  MoveL 1338 to (-196.6, 429.23, -4.47) mm, rotated rx 180 ry 0 rz -11.91 deg; joints [10.082, -29.328, 80.991, -91.112, 88.613, 140.802]
  MoveL 1339 to (-196.78, 429.13, -4.48) mm, rotated rx -180 ry 0 rz -11.91 deg; joints [10.077, -29.335, 81.007, -91.116, 88.609, 140.811]
  MoveL 1340 to (-196.95, 429.01, -4.47) mm, rotated rx -180 ry 0 rz -11.91 deg; joints [10.072, -29.343, 81.024, -91.12, 88.606, 140.82]
  MoveL 1341 to (-197.13, 428.87, -4.48) mm, rotated rx -180 ry 0 rz -11.91 deg; joints [10.066, -29.352, 81.044, -91.125, 88.604, 140.831]
  MoveL 1342 to (-197.37, 428.65, -4.48) mm, rotated rx 180 ry 0 rz -11.91 deg; joints [10.06, -29.366, 81.073, -91.13, 88.6, 140.847]
  MoveL 1343 to (-197.56, 428.44, -4.48) mm, rotated rx 180 ry 0 rz -11.91 deg; joints [10.055, -29.379, 81.102, -91.134, 88.597, 140.862]
  MoveL 1344 to (-197.72, 428.22, -4.48) mm, rotated rx -180 ry 0 rz -11.91 deg; joints [10.051, -29.391, 81.129, -91.138, 88.595, 140.877]
  MoveL 1345 to (-197.85, 428.01, -4.48) mm, rotated rx -180 ry 0 rz -11.91 deg; joints [10.048, -29.404, 81.157, -91.141, 88.593, 140.892]
  MoveL 1346 to (-197.98, 427.77, -4.48) mm, rotated rx 180 ry 0 rz -11.91 deg; joints [10.045, -29.418, 81.187, -91.143, 88.592, 140.909]
  MoveL 1347 to (-198.08, 427.53, -4.48) mm, rotated rx 180 ry 0 rz -11.91 deg; joints [10.043, -29.432, 81.217, -91.145, 88.591, 140.925]
  MoveL 1348 to (-198.16, 427.29, -4.48) mm, rotated rx 180 ry 0 rz -11.91 deg; joints [10.042, -29.445, 81.246, -91.146, 88.591, 140.94]
  MoveL 1349 to (-198.21, 427.04, -4.47) mm, rotated rx -180 ry 0 rz -11.91 deg; joints [10.042, -29.459, 81.275, -91.147, 88.591, 140.956]
  MoveL 1350 to (-198.25, 426.8, -4.48) mm, rotated rx -180 ry 0 rz -11.91 deg; joints [10.042, -29.472, 81.304, -91.147, 88.591, 140.971]
  MoveL 1351 to (-198.27, 426.56, -4.47) mm, rotated rx -180 ry 0 rz -11.91 deg; joints [10.043, -29.485, 81.332, -91.147, 88.592, 140.986]
  MoveL 1352 to (-198.27, 426.08, -4.48) mm, rotated rx -180 ry 0 rz -11.91 deg; joints [10.045, -29.51, 81.387, -91.146, 88.594, 141.016]
  MoveL 1353 to (-198.27, 425.59, -4.48) mm, rotated rx -180 ry 0 rz -11.91 deg; joints [10.048, -29.536, 81.442, -91.144, 88.597, 141.046]
  MoveL 1354 to (-198.25, 425.35, -4.47) mm, rotated rx -180 ry 0 rz -11.91 deg; joints [10.05, -29.549, 81.47, -91.143, 88.598, 141.061]
  MoveL 1355 to (-198.22, 425.11, -4.47) mm, rotated rx -180 ry 0 rz -11.91 deg; joints [10.053, -29.561, 81.497, -91.141, 88.6, 141.075]
  MoveL 1356 to (-198.16, 424.87, -4.48) mm, rotated rx -180 ry 0 rz -11.91 deg; joints [10.056, -29.573, 81.523, -91.139, 88.602, 141.089]
  MoveL 1357 to (-198.09, 424.63, -4.48) mm, rotated rx 180 ry 0 rz -11.91 deg; joints [10.06, -29.585, 81.549, -91.136, 88.605, 141.103]
  MoveL 1358 to (-197.99, 424.39, -4.48) mm, rotated rx 180 ry 0 rz -11.91 deg; joints [10.065, -29.597, 81.575, -91.133, 88.608, 141.117]
  MoveL 1359 to (-197.87, 424.15, -4.48) mm, rotated rx -180 ry 0 rz -11.91 deg; joints [10.07, -29.609, 81.6, -91.129, 88.612, 141.13]
  MoveL 1360 to (-197.73, 423.93, -4.47) mm, rotated rx -180 ry 0 rz -11.91 deg; joints [10.076, -29.619, 81.622, -91.125, 88.615, 141.142]
  MoveL 1361 to (-197.57, 423.71, -4.48) mm, rotated rx 180 ry 0 rz -11.91 deg; joints [10.083, -29.629, 81.644, -91.12, 88.62, 141.154]
  MoveL 1362 to (-197.38, 423.49, -4.48) mm, rotated rx -180 ry 0 rz -11.91 deg; joints [10.09, -29.639, 81.665, -91.114, 88.625, 141.165]
  MoveL 1363 to (-197.14, 423.27, -4.48) mm, rotated rx -180 ry 0 rz -11.91 deg; joints [10.099, -29.648, 81.685, -91.107, 88.631, 141.176]
  MoveL 1364 to (-196.96, 423.13, -4.48) mm, rotated rx -180 ry 0 rz -11.91 deg; joints [10.106, -29.654, 81.698, -91.102, 88.635, 141.182]
  MoveL 1365 to (-196.78, 423, -4.48) mm, rotated rx 180 ry 0 rz -11.91 deg; joints [10.113, -29.659, 81.708, -91.097, 88.639, 141.188]
  MoveL 1366 to (-196.6, 422.9, -4.48) mm, rotated rx -180 ry 0 rz -11.91 deg; joints [10.119, -29.663, 81.716, -91.092, 88.643, 141.192]
  MoveL 1367 to (-196.42, 422.81, -4.48) mm, rotated rx 180 ry 0 rz -11.91 deg; joints [10.126, -29.666, 81.723, -91.087, 88.647, 141.195]
  MoveL 1368 to (-196.18, 422.71, -4.48) mm, rotated rx -180 ry 0 rz -11.91 deg; joints [10.135, -29.669, 81.729, -91.08, 88.653, 141.199]
  MoveL 1369 to (-195.93, 422.63, -4.47) mm, rotated rx -180 ry 0 rz -11.91 deg; joints [10.143, -29.671, 81.733, -91.073, 88.658, 141.2]
  MoveL 1370 to (-195.69, 422.58, -4.48) mm, rotated rx 180 ry 0 rz -11.91 deg; joints [10.151, -29.671, 81.734, -91.067, 88.663, 141.201]
  MoveL 1371 to (-195.45, 422.54, -4.48) mm, rotated rx -180 ry 0 rz -11.91 deg; joints [10.159, -29.671, 81.733, -91.06, 88.668, 141.2]
  MoveL 1372 to (-195.21, 422.52, -4.48) mm, rotated rx 180 ry 0 rz -11.91 deg; joints [10.167, -29.67, 81.73, -91.054, 88.673, 141.199]
  MoveL 1373 to (-194.97, 422.52, -4.48) mm, rotated rx -180 ry 0 rz -11.91 deg; joints [10.175, -29.668, 81.726, -91.047, 88.678, 141.196]
  Set speed (38.1 mm/s)
  MoveL 1374 to (-194.97, 421.25, -4.48) mm, rotated rx -180 ry 0 rz -11.91 deg; joints [10.183, -29.735, 81.87, -91.043, 88.684, 141.274]
  MoveL 1375 to (-195.61, 421.25, -4.47) mm, rotated rx -180 ry 0 rz -11.91 deg; joints [10.162, -29.74, 81.883, -91.06, 88.671, 141.281]
  Set speed (25.4 mm/s)
  MoveL 1376 to (-195.61, 421.25, -6.84) mm, rotated rx 180 ry 0 rz -11.91 deg; joints [10.163, -29.63, 81.86, -91.062, 88.673, 141.368]
  MoveL 1377 to (-195.61, 421.89, -7.48) mm, rotated rx -180 ry 0 rz -11.91 deg; joints [10.159, -29.567, 81.781, -91.064, 88.67, 141.353]
  Set speed (38.1 mm/s)
  MoveL 1378 to (-194.97, 422.52, -7.47) mm, rotated rx 180 ry 0 rz -11.91 deg; joints [10.176, -29.527, 81.696, -91.05, 88.68, 141.306]
  Set speed (76.2 mm/s)
  MoveL 1379 to (213.41, 422.52, -7.47) mm, rotated rx -180 ry 0 rz -11.91 deg; joints [22.898, -22.659, 66.695, -81.959, 97.664, 133.746]
  MoveL 1380 to (213.89, 422.53, -7.47) mm, rotated rx -180 ry 0 rz -11.91 deg; joints [22.912, -22.646, 66.667, -81.951, 97.676, 133.732]
  MoveL 1381 to (214.13, 422.55, -7.48) mm, rotated rx 180 ry 0 rz -11.91 deg; joints [22.919, -22.638, 66.651, -81.948, 97.682, 133.724]
  MoveL 1382 to (214.37, 422.59, -7.48) mm, rotated rx 180 ry 0 rz -11.91 deg; joints [22.925, -22.629, 66.632, -81.945, 97.688, 133.715]
  MoveL 1383 to (214.61, 422.65, -7.48) mm, rotated rx -180 ry 0 rz -11.91 deg; joints [22.931, -22.619, 66.61, -81.942, 97.694, 133.704]
  MoveL 1384 to (214.85, 422.74, -7.47) mm, rotated rx -180 ry 0 rz -11.91 deg; joints [22.937, -22.608, 66.586, -81.939, 97.7, 133.692]
  MoveL 1385 to (215.09, 422.84, -7.48) mm, rotated rx 180 ry 0 rz -11.91 deg; joints [22.943, -22.595, 66.558, -81.937, 97.706, 133.678]
  MoveL 1386 to (215.34, 422.97, -7.48) mm, rotated rx 180 ry 0 rz -11.91 deg; joints [22.948, -22.58, 66.527, -81.936, 97.712, 133.662]
  MoveL 1387 to (215.58, 423.13, -7.48) mm, rotated rx -180 ry 0 rz -11.91 deg; joints [22.953, -22.564, 66.493, -81.935, 97.718, 133.644]
  MoveL 1388 to (215.82, 423.33, -7.48) mm, rotated rx -180 ry 0 rz -11.91 deg; joints [22.958, -22.546, 66.454, -81.934, 97.724, 133.624]
  MoveL 1389 to (215.96, 423.46, -7.47) mm, rotated rx -180 ry 0 rz -11.91 deg; joints [22.96, -22.533, 66.428, -81.934, 97.728, 133.61]
  MoveL 1390 to (216.09, 423.6, -7.48) mm, rotated rx 180 ry 0 rz -11.91 deg; joints [22.962, -22.522, 66.403, -81.935, 97.731, 133.597]
  MoveL 1391 to (216.2, 423.73, -7.48) mm, rotated rx 180 ry 0 rz -11.91 deg; joints [22.964, -22.51, 66.379, -81.935, 97.734, 133.585]
  MoveL 1392 to (216.3, 423.87, -7.48) mm, rotated rx -180 ry 0 rz -11.91 deg; joints [22.965, -22.499, 66.355, -81.936, 97.737, 133.573]
  MoveL 1393 to (216.39, 424.01, -7.48) mm, rotated rx -180 ry 0 rz -11.91 deg; joints [22.966, -22.488, 66.331, -81.937, 97.739, 133.56]
  MoveL 1394 to (216.47, 424.15, -7.48) mm, rotated rx -180 ry 0 rz -11.91 deg; joints [22.967, -22.477, 66.308, -81.938, 97.741, 133.548]
  MoveL 1395 to (216.6, 424.39, -7.48) mm, rotated rx -180 ry 0 rz -11.91 deg; joints [22.967, -22.459, 66.27, -81.94, 97.745, 133.528]
  MoveL 1396 to (216.69, 424.63, -7.48) mm, rotated rx -180 ry 0 rz -11.91 deg; joints [22.967, -22.441, 66.232, -81.943, 97.747, 133.508]
  MoveL 1397 to (216.77, 424.87, -7.47) mm, rotated rx 180 ry 0 rz -11.91 deg; joints [22.966, -22.424, 66.196, -81.946, 97.749, 133.489]
  MoveL 1398 to (216.82, 425.11, -7.47) mm, rotated rx -180 ry 0 rz -11.91 deg; joints [22.965, -22.407, 66.16, -81.95, 97.751, 133.47]
  MoveL 1399 to (216.86, 425.35, -7.47) mm, rotated rx -180 ry 0 rz -11.91 deg; joints [22.963, -22.391, 66.126, -81.954, 97.752, 133.452]
  MoveL 1400 to (216.88, 425.59, -7.48) mm, rotated rx 180 ry 0 rz -11.91 deg; joints [22.96, -22.376, 66.093, -81.958, 97.753, 133.434]
  MoveL 1401 to (216.88, 426.08, -7.48) mm, rotated rx -180 ry 0 rz -11.91 deg; joints [22.955, -22.345, 66.029, -81.966, 97.753, 133.4]
  MoveL 1402 to (216.88, 427.04, -7.48) mm, rotated rx -180 ry 0 rz -11.91 deg; joints [22.943, -22.284, 65.9, -81.984, 97.754, 133.331]
  MoveL 1403 to (216.86, 427.29, -7.47) mm, rotated rx 180 ry 0 rz -11.91 deg; joints [22.939, -22.269, 65.869, -81.989, 97.754, 133.314]
  MoveL 1404 to (216.83, 427.53, -7.48) mm, rotated rx -180 ry 0 rz -11.91 deg; joints [22.935, -22.255, 65.838, -81.993, 97.754, 133.297]
  MoveL 1405 to (216.78, 427.77, -7.48) mm, rotated rx -180 ry 0 rz -11.91 deg; joints [22.931, -22.241, 65.809, -81.999, 97.753, 133.282]
  MoveL 1406 to (216.71, 428.01, -7.48) mm, rotated rx -180 ry 0 rz -11.91 deg; joints [22.926, -22.228, 65.781, -82.004, 97.751, 133.266]
  MoveL 1407 to (216.63, 428.21, -7.48) mm, rotated rx 180 ry 0 rz -11.91 deg; joints [22.921, -22.217, 65.759, -82.009, 97.749, 133.254]
  MoveL 1408 to (216.54, 428.41, -7.48) mm, rotated rx -180 ry 0 rz -11.91 deg; joints [22.916, -22.207, 65.737, -82.014, 97.747, 133.242]
  MoveL 1409 to (216.43, 428.61, -7.48) mm, rotated rx 180 ry 0 rz -11.91 deg; joints [22.911, -22.197, 65.717, -82.019, 97.745, 133.231]
  MoveL 1410 to (216.3, 428.81, -7.48) mm, rotated rx 180 ry 0 rz -11.91 deg; joints [22.904, -22.188, 65.697, -82.025, 97.742, 133.22]
  MoveL 1411 to (216.16, 428.99, -7.48) mm, rotated rx 180 ry 0 rz -11.91 deg; joints [22.898, -22.18, 65.681, -82.031, 97.738, 133.211]
  MoveL 1412 to (215.99, 429.18, -7.47) mm, rotated rx -180 ry 0 rz -11.91 deg; joints [22.891, -22.173, 65.665, -82.037, 97.735, 133.202]
  MoveL 1413 to (215.78, 429.38, -7.48) mm, rotated rx -180 ry 0 rz -11.91 deg; joints [22.883, -22.165, 65.65, -82.044, 97.729, 133.193]
  MoveL 1414 to (215.57, 429.55, -7.48) mm, rotated rx -180 ry 0 rz -11.91 deg; joints [22.874, -22.16, 65.64, -82.05, 97.724, 133.187]
  MoveL 1415 to (215.39, 429.67, -7.47) mm, rotated rx -180 ry 0 rz -11.91 deg; joints [22.868, -22.157, 65.633, -82.055, 97.72, 133.183]
  MoveL 1416 to (215.21, 429.78, -7.48) mm, rotated rx -180 ry 0 rz -11.91 deg; joints [22.861, -22.155, 65.63, -82.06, 97.716, 133.181]
  MoveL 1417 to (215.02, 429.87, -7.48) mm, rotated rx 180 ry 0 rz -11.91 deg; joints [22.855, -22.154, 65.628, -82.065, 97.711, 133.179]
  MoveL 1418 to (214.84, 429.94, -7.47) mm, rotated rx -180 ry 0 rz -11.91 deg; joints [22.849, -22.154, 65.628, -82.069, 97.707, 133.179]
  MoveL 1419 to (214.61, 430.02, -7.48) mm, rotated rx 180 ry 0 rz -11.91 deg; joints [22.841, -22.156, 65.63, -82.074, 97.701, 133.179]
  MoveL 1420 to (214.37, 430.08, -7.48) mm, rotated rx -180 ry 0 rz -11.91 deg; joints [22.833, -22.158, 65.636, -82.079, 97.695, 133.181]
  MoveL 1421 to (214.13, 430.13, -7.47) mm, rotated rx -180 ry 0 rz -11.91 deg; joints [22.826, -22.162, 65.644, -82.084, 97.689, 133.185]
  MoveL 1422 to (213.89, 430.15, -7.48) mm, rotated rx -180 ry 0 rz -11.91 deg; joints [22.819, -22.166, 65.654, -82.088, 97.683, 133.19]
  MoveL 1423 to (213.41, 430.15, -7.48) mm, rotated rx -180 ry 0 rz -11.91 deg; joints [22.805, -22.179, 65.681, -82.096, 97.671, 133.203]
  MoveL 1424 to (-194.49, 430.15, -7.47) mm, rotated rx 180 ry 0 rz -11.91 deg; joints [10.147, -29.119, 80.811, -91.062, 88.653, 140.83]
  MoveL 1425 to (-195.36, 430.14, -7.48) mm, rotated rx 180 ry 0 rz -11.91 deg; joints [10.118, -29.128, 80.83, -91.084, 88.636, 140.841]
  MoveL 1426 to (-195.58, 430.12, -7.48) mm, rotated rx -180 ry 0 rz -11.91 deg; joints [10.111, -29.131, 80.837, -91.09, 88.631, 140.845]
  MoveL 1427 to (-195.8, 430.08, -7.47) mm, rotated rx 180 ry 0 rz -11.91 deg; joints [10.104, -29.136, 80.847, -91.096, 88.627, 140.85]
  MoveL 1428 to (-196.02, 430.02, -7.48) mm, rotated rx -180 ry 0 rz -11.91 deg; joints [10.097, -29.141, 80.858, -91.101, 88.623, 140.856]
  MoveL 1429 to (-196.24, 429.94, -7.47) mm, rotated rx 180 ry 0 rz -11.91 deg; joints [10.09, -29.147, 80.871, -91.107, 88.619, 140.863]
  MoveL 1430 to (-196.42, 429.87, -7.48) mm, rotated rx -180 ry 0 rz -11.91 deg; joints [10.085, -29.152, 80.884, -91.111, 88.616, 140.87]
  MoveL 1431 to (-196.56, 429.8, -7.48) mm, rotated rx -180 ry 0 rz -11.91 deg; joints [10.08, -29.158, 80.895, -91.115, 88.613, 140.876]
  MoveL 1432 to (-196.71, 429.71, -7.48) mm, rotated rx 180 ry 0 rz -11.91 deg; joints [10.076, -29.163, 80.907, -91.118, 88.61, 140.883]
  MoveL 1433 to (-196.86, 429.62, -7.47) mm, rotated rx 180 ry 0 rz -11.91 deg; joints [10.072, -29.17, 80.921, -91.122, 88.608, 140.891]
  MoveL 1434 to (-197.01, 429.52, -7.47) mm, rotated rx 180 ry 0 rz -11.91 deg; joints [10.067, -29.176, 80.936, -91.125, 88.605, 140.899]
  MoveL 1435 to (-197.15, 429.4, -7.48) mm, rotated rx -180 ry 0 rz -11.91 deg; joints [10.063, -29.184, 80.953, -91.129, 88.603, 140.908]
  MoveL 1436 to (-197.3, 429.27, -7.48) mm, rotated rx -180 ry 0 rz -11.91 deg; joints [10.059, -29.192, 80.971, -91.132, 88.601, 140.918]
  MoveL 1437 to (-197.46, 429.1, -7.48) mm, rotated rx 180 ry 0 rz -11.91 deg; joints [10.055, -29.203, 80.993, -91.136, 88.598, 140.93]
  MoveL 1438 to (-197.6, 428.94, -7.48) mm, rotated rx -180 ry 0 rz -11.91 deg; joints [10.051, -29.213, 81.015, -91.139, 88.596, 140.942]
  MoveL 1439 to (-197.76, 428.71, -7.48) mm, rotated rx -180 ry 0 rz -11.91 deg; joints [10.047, -29.226, 81.045, -91.143, 88.594, 140.958]
  MoveL 1440 to (-197.9, 428.47, -7.48) mm, rotated rx -180 ry 0 rz -11.91 deg; joints [10.044, -29.24, 81.074, -91.146, 88.593, 140.974]
  MoveL 1441 to (-198.01, 428.24, -7.48) mm, rotated rx 180 ry 0 rz -11.91 deg; joints [10.042, -29.253, 81.103, -91.148, 88.591, 140.989]
  MoveL 1442 to (-198.1, 428.01, -7.48) mm, rotated rx 180 ry 0 rz -11.91 deg; joints [10.04, -29.266, 81.132, -91.149, 88.591, 141.005]
  MoveL 1443 to (-198.17, 427.77, -7.48) mm, rotated rx -180 ry 0 rz -11.91 deg; joints [10.039, -29.28, 81.161, -91.151, 88.591, 141.021]
  MoveL 1444 to (-198.23, 427.53, -7.47) mm, rotated rx -180 ry 0 rz -11.91 deg; joints [10.039, -29.293, 81.19, -91.151, 88.591, 141.036]
  MoveL 1445 to (-198.26, 427.29, -7.47) mm, rotated rx -180 ry 0 rz -11.91 deg; joints [10.039, -29.306, 81.218, -91.151, 88.591, 141.051]
  MoveL 1446 to (-198.27, 427.04, -7.47) mm, rotated rx -180 ry 0 rz -11.91 deg; joints [10.04, -29.319, 81.246, -91.151, 88.592, 141.067]
  MoveL 1447 to (-198.27, 426.08, -7.48) mm, rotated rx -180 ry 0 rz -11.91 deg; joints [10.046, -29.37, 81.357, -91.148, 88.597, 141.126]
  MoveL 1448 to (-198.27, 425.59, -7.48) mm, rotated rx 180 ry 0 rz -11.91 deg; joints [10.049, -29.396, 81.412, -91.146, 88.599, 141.156]
  MoveL 1449 to (-198.25, 425.35, -7.48) mm, rotated rx 180 ry 0 rz -11.91 deg; joints [10.051, -29.408, 81.44, -91.145, 88.601, 141.171]
  MoveL 1450 to (-198.22, 425.11, -7.48) mm, rotated rx -180 ry 0 rz -11.91 deg; joints [10.053, -29.421, 81.466, -91.143, 88.603, 141.185]
  MoveL 1451 to (-198.16, 424.87, -7.48) mm, rotated rx -180 ry 0 rz -11.91 deg; joints [10.057, -29.433, 81.493, -91.141, 88.605, 141.199]
  MoveL 1452 to (-198.09, 424.63, -7.48) mm, rotated rx 180 ry 0 rz -11.91 deg; joints [10.061, -29.445, 81.519, -91.138, 88.608, 141.213]
  MoveL 1453 to (-197.99, 424.39, -7.47) mm, rotated rx -180 ry 0 rz -11.91 deg; joints [10.065, -29.457, 81.545, -91.135, 88.611, 141.227]
  MoveL 1454 to (-197.87, 424.15, -7.48) mm, rotated rx 180 ry 0 rz -11.91 deg; joints [10.071, -29.469, 81.57, -91.131, 88.614, 141.24]
  MoveL 1455 to (-197.73, 423.93, -7.48) mm, rotated rx -180 ry 0 rz -11.91 deg; joints [10.077, -29.479, 81.592, -91.127, 88.618, 141.252]
  MoveL 1456 to (-197.57, 423.71, -7.48) mm, rotated rx -180 ry 0 rz -11.91 deg; joints [10.083, -29.489, 81.614, -91.122, 88.622, 141.264]
  MoveL 1457 to (-197.38, 423.49, -7.47) mm, rotated rx -180 ry 0 rz -11.91 deg; joints [10.091, -29.499, 81.635, -91.116, 88.627, 141.275]
  MoveL 1458 to (-197.14, 423.27, -7.47) mm, rotated rx -180 ry 0 rz -11.91 deg; joints [10.1, -29.508, 81.655, -91.109, 88.633, 141.286]
  MoveL 1459 to (-196.96, 423.13, -7.48) mm, rotated rx -180 ry 0 rz -11.91 deg; joints [10.107, -29.514, 81.668, -91.104, 88.637, 141.293]
  MoveL 1460 to (-196.78, 423, -7.47) mm, rotated rx -180 ry 0 rz -11.91 deg; joints [10.113, -29.519, 81.678, -91.099, 88.642, 141.298]
  MoveL 1461 to (-196.6, 422.9, -7.48) mm, rotated rx -180 ry 0 rz -11.91 deg; joints [10.12, -29.523, 81.686, -91.094, 88.646, 141.302]
  MoveL 1462 to (-196.42, 422.81, -7.48) mm, rotated rx 180 ry 0 rz -11.91 deg; joints [10.127, -29.526, 81.693, -91.089, 88.65, 141.306]
  MoveL 1463 to (-196.18, 422.71, -7.48) mm, rotated rx -180 ry 0 rz -11.91 deg; joints [10.135, -29.529, 81.699, -91.082, 88.655, 141.309]
  MoveL 1464 to (-195.93, 422.63, -7.47) mm, rotated rx -180 ry 0 rz -11.91 deg; joints [10.144, -29.53, 81.703, -91.075, 88.66, 141.311]
  MoveL 1465 to (-195.69, 422.58, -7.48) mm, rotated rx -180 ry 0 rz -11.91 deg; joints [10.152, -29.531, 81.704, -91.069, 88.665, 141.311]
  MoveL 1466 to (-195.45, 422.54, -7.48) mm, rotated rx -180 ry 0 rz -11.91 deg; joints [10.16, -29.531, 81.703, -91.062, 88.67, 141.311]
  MoveL 1467 to (-195.21, 422.52, -7.48) mm, rotated rx -180 ry 0 rz -11.91 deg; joints [10.168, -29.53, 81.7, -91.056, 88.675, 141.309]
  MoveL 1468 to (-194.97, 422.52, -7.47) mm, rotated rx 180 ry 0 rz -11.91 deg; joints [10.176, -29.527, 81.696, -91.05, 88.68, 141.306]
  Set speed (38.1 mm/s)
  MoveL 1469 to (-194.97, 421.25, -7.48) mm, rotated rx -180 ry 0 rz -11.91 deg; joints [10.184, -29.594, 81.84, -91.045, 88.686, 141.384]
  MoveL 1470 to (-195.61, 421.25, -7.47) mm, rotated rx -180 ry 0 rz -11.91 deg; joints [10.163, -29.6, 81.853, -91.062, 88.674, 141.392]
  Set speed (25.4 mm/s)
  MoveL 1471 to (-195.61, 421.25, -9.84) mm, rotated rx -180 ry 0 rz -11.91 deg; joints [10.163, -29.489, 81.829, -91.064, 88.675, 141.478]
  MoveL 1472 to (-195.61, 421.89, -10.48) mm, rotated rx -180 ry 0 rz -11.91 deg; joints [10.16, -29.426, 81.75, -91.066, 88.673, 141.463]
  Set speed (38.1 mm/s)
  MoveL 1473 to (-194.97, 422.52, -10.48) mm, rotated rx 180 ry 0 rz -11.91 deg; joints [10.177, -29.387, 81.665, -91.052, 88.683, 141.416]
  Set speed (76.2 mm/s)
  MoveL 1474 to (213.41, 422.52, -10.48) mm, rotated rx -180 ry 0 rz -11.91 deg; joints [22.899, -22.526, 66.66, -81.946, 97.651, 133.844]
  MoveL 1475 to (213.89, 422.53, -10.47) mm, rotated rx -180 ry 0 rz -11.91 deg; joints [22.913, -22.513, 66.632, -81.938, 97.663, 133.83]
  MoveL 1476 to (214.13, 422.55, -10.48) mm, rotated rx -180 ry 0 rz -11.91 deg; joints [22.919, -22.505, 66.616, -81.934, 97.669, 133.822]
  MoveL 1477 to (214.37, 422.59, -10.47) mm, rotated rx 180 ry 0 rz -11.91 deg; joints [22.926, -22.496, 66.597, -81.931, 97.675, 133.813]
  MoveL 1478 to (214.61, 422.65, -10.48) mm, rotated rx -180 ry 0 rz -11.91 deg; joints [22.932, -22.486, 66.575, -81.928, 97.681, 133.802]
  MoveL 1479 to (214.85, 422.74, -10.48) mm, rotated rx -180 ry 0 rz -11.91 deg; joints [22.938, -22.475, 66.551, -81.926, 97.687, 133.79]
  MoveL 1480 to (215.09, 422.84, -10.48) mm, rotated rx -180 ry 0 rz -11.91 deg; joints [22.944, -22.462, 66.523, -81.923, 97.693, 133.776]
  MoveL 1481 to (215.34, 422.97, -10.48) mm, rotated rx -180 ry 0 rz -11.91 deg; joints [22.949, -22.448, 66.493, -81.922, 97.699, 133.76]
  MoveL 1482 to (215.58, 423.13, -10.48) mm, rotated rx 180 ry 0 rz -11.91 deg; joints [22.954, -22.431, 66.458, -81.921, 97.705, 133.742]
  MoveL 1483 to (215.82, 423.33, -10.47) mm, rotated rx -180 ry 0 rz -11.91 deg; joints [22.959, -22.413, 66.419, -81.92, 97.711, 133.722]
  MoveL 1484 to (215.96, 423.46, -10.47) mm, rotated rx -180 ry 0 rz -11.91 deg; joints [22.961, -22.401, 66.393, -81.92, 97.715, 133.708]
  MoveL 1485 to (216.09, 423.6, -10.48) mm, rotated rx -180 ry 0 rz -11.91 deg; joints [22.963, -22.389, 66.368, -81.921, 97.718, 133.695]
  MoveL 1486 to (216.2, 423.73, -10.48) mm, rotated rx 180 ry 0 rz -11.91 deg; joints [22.965, -22.378, 66.344, -81.921, 97.721, 133.683]
  MoveL 1487 to (216.3, 423.87, -10.48) mm, rotated rx -180 ry 0 rz -11.91 deg; joints [22.966, -22.366, 66.32, -81.922, 97.724, 133.67]
  MoveL 1488 to (216.39, 424.01, -10.48) mm, rotated rx -180 ry 0 rz -11.91 deg; joints [22.967, -22.355, 66.296, -81.923, 97.726, 133.658]
  MoveL 1489 to (216.47, 424.15, -10.48) mm, rotated rx -180 ry 0 rz -11.91 deg; joints [22.968, -22.344, 66.273, -81.924, 97.728, 133.646]
  MoveL 1490 to (216.69, 424.27, -10.47) mm, rotated rx -180 ry 0 rz -11.91 deg; joints [22.972, -22.331, 66.245, -81.923, 97.734, 133.631]
  MoveL 1491 to (219.83, 424.27, -10.48) mm, rotated rx -180 ry 0 rz -11.91 deg; joints [23.063, -22.249, 66.068, -81.872, 97.812, 133.546]
  MoveL 1492 to (220.05, 424.15, -10.47) mm, rotated rx -180 ry 0 rz -11.91 deg; joints [23.071, -22.25, 66.071, -81.866, 97.817, 133.548]
  MoveL 1493 to (220.05, 53.41, -10.48) mm, rotated rx 180 ry 0 rz -11.91 deg; joints [28.668, -39.388, 103.529, -74.583, 96.903, 154.267]
  MoveL 1494 to (219.83, 53.18, -10.47) mm, rotated rx -180 ry 0 rz -11.91 deg; joints [28.664, -39.401, 103.558, -74.584, 96.897, 154.283]
  MoveL 1495 to (-199.12, 53.17, -10.48) mm, rotated rx 180 ry 0 rz -11.91 deg; joints [12.81, -44.761, 116.802, -88.93, 89.927, 161.175]
  MoveL 1496 to (-199.7, 53.18, -10.47) mm, rotated rx -180 ry 0 rz -11.91 deg; joints [12.785, -44.765, 116.813, -88.953, 89.92, 161.182]
  MoveL 1497 to (-199.9, 53.41, -10.48) mm, rotated rx 180 ry 0 rz -11.91 deg; joints [12.775, -44.759, 116.797, -88.963, 89.917, 161.172]
  MoveL 1498 to (-199.9, 424.15, -10.48) mm, rotated rx -180 ry 0 rz -11.91 deg; joints [10.004, -29.346, 81.58, -91.187, 88.576, 141.374]
  MoveL 1499 to (-199.7, 424.27, -10.47) mm, rotated rx -180 ry 0 rz -11.91 deg; joints [10.01, -29.338, 81.562, -91.182, 88.58, 141.364]
  MoveL 1500 to (-198.11, 424.27, -10.47) mm, rotated rx -180 ry 0 rz -11.91 deg; joints [10.063, -29.324, 81.53, -91.14, 88.611, 141.346]
  MoveL 1501 to (-197.87, 424.15, -10.48) mm, rotated rx -180 ry 0 rz -11.91 deg; joints [10.071, -29.328, 81.539, -91.133, 88.617, 141.35]
  MoveL 1502 to (-197.73, 423.93, -10.48) mm, rotated rx -180 ry 0 rz -11.91 deg; joints [10.077, -29.338, 81.561, -91.129, 88.621, 141.362]
  MoveL 1503 to (-197.57, 423.71, -10.48) mm, rotated rx -180 ry 0 rz -11.91 deg; joints [10.084, -29.348, 81.583, -91.124, 88.625, 141.374]
  MoveL 1504 to (-197.38, 423.49, -10.48) mm, rotated rx -180 ry 0 rz -11.91 deg; joints [10.092, -29.358, 81.604, -91.118, 88.63, 141.385]
  MoveL 1505 to (-197.14, 423.27, -10.48) mm, rotated rx -180 ry 0 rz -11.91 deg; joints [10.101, -29.368, 81.624, -91.111, 88.636, 141.396]
  MoveL 1506 to (-196.96, 423.13, -10.48) mm, rotated rx -180 ry 0 rz -11.91 deg; joints [10.107, -29.373, 81.637, -91.106, 88.64, 141.402]
  MoveL 1507 to (-196.78, 423, -10.48) mm, rotated rx -180 ry 0 rz -11.91 deg; joints [10.114, -29.378, 81.647, -91.101, 88.644, 141.408]
  MoveL 1508 to (-196.6, 422.9, -10.48) mm, rotated rx 180 ry 0 rz -11.91 deg; joints [10.121, -29.382, 81.655, -91.096, 88.648, 141.412]
  MoveL 1509 to (-196.42, 422.81, -10.48) mm, rotated rx -180 ry 0 rz -11.91 deg; joints [10.127, -29.385, 81.662, -91.091, 88.652, 141.415]
  MoveL 1510 to (-196.18, 422.71, -10.47) mm, rotated rx -180 ry 0 rz -11.91 deg; joints [10.136, -29.388, 81.668, -91.084, 88.658, 141.419]
  MoveL 1511 to (-195.93, 422.63, -10.47) mm, rotated rx -180 ry 0 rz -11.91 deg; joints [10.144, -29.39, 81.672, -91.077, 88.663, 141.421]
  MoveL 1512 to (-195.69, 422.58, -10.48) mm, rotated rx 180 ry 0 rz -11.91 deg; joints [10.153, -29.39, 81.673, -91.071, 88.668, 141.421]
  MoveL 1513 to (-195.45, 422.54, -10.48) mm, rotated rx -180 ry 0 rz -11.91 deg; joints [10.161, -29.39, 81.673, -91.064, 88.673, 141.421]
  MoveL 1514 to (-195.21, 422.52, -10.48) mm, rotated rx 180 ry 0 rz -11.91 deg; joints [10.169, -29.389, 81.67, -91.058, 88.678, 141.419]
  MoveL 1515 to (-194.97, 422.52, -10.48) mm, rotated rx 180 ry 0 rz -11.91 deg; joints [10.177, -29.387, 81.665, -91.052, 88.683, 141.416]
  Set speed (38.1 mm/s)
  MoveL 1516 to (-194.97, 421.25, -10.48) mm, rotated rx -180 ry 0 rz -11.91 deg; joints [10.184, -29.453, 81.81, -91.047, 88.689, 141.494]
  MoveL 1517 to (-195.61, 421.25, -10.48) mm, rotated rx -180 ry 0 rz -11.91 deg; joints [10.163, -29.459, 81.823, -91.064, 88.676, 141.502]
  Set speed (25.4 mm/s)
  MoveL 1518 to (-195.61, 421.25, -12.84) mm, rotated rx -180 ry 0 rz -11.91 deg; joints [10.164, -29.348, 81.798, -91.066, 88.678, 141.588]
  MoveL 1519 to (-195.61, 421.89, -13.48) mm, rotated rx -180 ry 0 rz -11.91 deg; joints [10.16, -29.285, 81.719, -91.068, 88.675, 141.572]
  Set speed (38.1 mm/s)
  MoveL 1520 to (-194.97, 422.52, -13.48) mm, rotated rx 180 ry 0 rz -11.91 deg; joints [10.177, -29.246, 81.633, -91.054, 88.685, 141.526]
  Set speed (76.2 mm/s)
  MoveL 1521 to (213.41, 422.52, -13.48) mm, rotated rx 180 ry 0 rz -11.91 deg; joints [22.9, -22.393, 66.624, -81.932, 97.638, 133.941]
  MoveL 1522 to (213.89, 422.53, -13.47) mm, rotated rx -180 ry 0 rz -11.91 deg; joints [22.914, -22.38, 66.597, -81.924, 97.65, 133.928]
  MoveL 1523 to (214.13, 422.55, -13.47) mm, rotated rx -180 ry 0 rz -11.91 deg; joints [22.92, -22.372, 66.58, -81.92, 97.656, 133.92]
  MoveL 1524 to (214.37, 422.59, -13.47) mm, rotated rx 180 ry 0 rz -11.91 deg; joints [22.927, -22.363, 66.561, -81.917, 97.662, 133.91]
  MoveL 1525 to (214.61, 422.65, -13.48) mm, rotated rx -180 ry 0 rz -11.91 deg; joints [22.933, -22.353, 66.539, -81.914, 97.668, 133.899]
  MoveL 1526 to (214.85, 422.74, -13.47) mm, rotated rx -180 ry 0 rz -11.91 deg; joints [22.939, -22.342, 66.515, -81.912, 97.674, 133.887]
  MoveL 1527 to (215.09, 422.84, -13.48) mm, rotated rx -180 ry 0 rz -11.91 deg; joints [22.945, -22.329, 66.488, -81.91, 97.68, 133.873]
  MoveL 1528 to (215.34, 422.97, -13.48) mm, rotated rx 180 ry 0 rz -11.91 deg; joints [22.95, -22.314, 66.457, -81.908, 97.686, 133.857]
  MoveL 1529 to (215.58, 423.13, -13.47) mm, rotated rx -180 ry 0 rz -11.91 deg; joints [22.955, -22.298, 66.422, -81.907, 97.692, 133.839]
  MoveL 1530 to (215.82, 423.33, -13.47) mm, rotated rx -180 ry 0 rz -11.91 deg; joints [22.96, -22.28, 66.383, -81.907, 97.698, 133.819]
  MoveL 1531 to (215.96, 423.46, -13.48) mm, rotated rx -180 ry 0 rz -11.91 deg; joints [22.962, -22.268, 66.357, -81.907, 97.702, 133.806]
  MoveL 1532 to (216.09, 423.6, -13.48) mm, rotated rx 180 ry 0 rz -11.91 deg; joints [22.964, -22.256, 66.332, -81.907, 97.705, 133.793]
  MoveL 1533 to (216.2, 423.73, -13.47) mm, rotated rx -180 ry 0 rz -11.91 deg; joints [22.966, -22.244, 66.308, -81.908, 97.708, 133.78]
  MoveL 1534 to (216.3, 423.87, -13.48) mm, rotated rx 180 ry 0 rz -11.91 deg; joints [22.967, -22.233, 66.284, -81.908, 97.711, 133.768]
  MoveL 1535 to (216.39, 424.01, -13.48) mm, rotated rx 180 ry 0 rz -11.91 deg; joints [22.968, -22.222, 66.261, -81.909, 97.713, 133.755]
  MoveL 1536 to (216.47, 424.15, -13.47) mm, rotated rx 180 ry 0 rz -11.91 deg; joints [22.968, -22.211, 66.238, -81.911, 97.715, 133.743]
  MoveL 1537 to (216.69, 424.27, -13.47) mm, rotated rx -180 ry 0 rz -11.91 deg; joints [22.973, -22.198, 66.209, -81.909, 97.721, 133.729]
  MoveL 1538 to (219.83, 424.27, -13.48) mm, rotated rx 180 ry 0 rz -11.91 deg; joints [23.064, -22.116, 66.032, -81.858, 97.799, 133.643]
  MoveL 1539 to (220.05, 424.15, -13.47) mm, rotated rx 180 ry 0 rz -11.91 deg; joints [23.072, -22.117, 66.035, -81.852, 97.804, 133.645]
  MoveL 1540 to (220.05, 53.41, -13.48) mm, rotated rx -180 ry 0 rz -11.91 deg; joints [28.669, -39.225, 103.499, -74.566, 96.868, 154.397]
  MoveL 1541 to (219.83, 53.18, -13.47) mm, rotated rx -180 ry 0 rz -11.91 deg; joints [28.665, -39.238, 103.529, -74.567, 96.862, 154.412]
  MoveL 1542 to (-197.29, 53.18, -13.48) mm, rotated rx -180 ry 0 rz -11.91 deg; joints [12.887, -44.563, 116.736, -88.857, 89.949, 161.308]
  MoveL 1543 to (-197.94, 53.18, -13.47) mm, rotated rx -180 ry 0 rz -11.91 deg; joints [12.86, -44.568, 116.748, -88.883, 89.94, 161.315]
  MoveL 1544 to (-198.16, 53.41, -13.47) mm, rotated rx -180 ry 0 rz -11.91 deg; joints [12.848, -44.561, 116.733, -88.894, 89.937, 161.306]
  MoveL 1545 to (-198.16, 424.15, -13.48) mm, rotated rx -180 ry 0 rz -11.91 deg; joints [10.062, -29.19, 81.513, -91.143, 88.614, 141.463]
  MoveL 1546 to (-198.01, 424.27, -13.47) mm, rotated rx -180 ry 0 rz -11.91 deg; joints [10.067, -29.182, 81.496, -91.14, 88.616, 141.454]
  MoveL 1547 to (-197.87, 424.15, -13.47) mm, rotated rx 180 ry 0 rz -11.91 deg; joints [10.072, -29.187, 81.507, -91.135, 88.619, 141.459]
  MoveL 1548 to (-197.73, 423.93, -13.48) mm, rotated rx -180 ry 0 rz -11.91 deg; joints [10.078, -29.197, 81.53, -91.131, 88.623, 141.471]
  MoveL 1549 to (-197.57, 423.71, -13.47) mm, rotated rx -180 ry 0 rz -11.91 deg; joints [10.084, -29.207, 81.551, -91.126, 88.627, 141.483]
  MoveL 1550 to (-197.38, 423.49, -13.47) mm, rotated rx -180 ry 0 rz -11.91 deg; joints [10.092, -29.217, 81.573, -91.12, 88.632, 141.494]
  MoveL 1551 to (-197.22, 423.33, -13.48) mm, rotated rx -180 ry 0 rz -11.91 deg; joints [10.098, -29.224, 81.587, -91.116, 88.636, 141.502]
  MoveL 1552 to (-197.14, 423.27, -13.47) mm, rotated rx -180 ry 0 rz -11.91 deg; joints [10.101, -29.227, 81.593, -91.113, 88.638, 141.505]
  MoveL 1553 to (-196.96, 423.13, -13.48) mm, rotated rx -180 ry 0 rz -11.91 deg; joints [10.108, -29.232, 81.605, -91.108, 88.642, 141.512]
  MoveL 1554 to (-196.78, 423, -13.47) mm, rotated rx -180 ry 0 rz -11.91 deg; joints [10.115, -29.237, 81.615, -91.103, 88.647, 141.517]
  MoveL 1555 to (-196.6, 422.9, -13.48) mm, rotated rx -180 ry 0 rz -11.91 deg; joints [10.121, -29.241, 81.624, -91.098, 88.651, 141.521]
  MoveL 1556 to (-196.42, 422.81, -13.48) mm, rotated rx -180 ry 0 rz -11.91 deg; joints [10.128, -29.244, 81.63, -91.093, 88.655, 141.525]
  MoveL 1557 to (-196.18, 422.71, -13.48) mm, rotated rx 180 ry 0 rz -11.91 deg; joints [10.136, -29.247, 81.637, -91.086, 88.66, 141.528]
  MoveL 1558 to (-195.93, 422.63, -13.48) mm, rotated rx 180 ry 0 rz -11.91 deg; joints [10.145, -29.249, 81.64, -91.079, 88.665, 141.53]
  MoveL 1559 to (-195.69, 422.58, -13.48) mm, rotated rx 180 ry 0 rz -11.91 deg; joints [10.153, -29.249, 81.642, -91.073, 88.67, 141.531]
  MoveL 1560 to (-195.45, 422.54, -13.47) mm, rotated rx -180 ry 0 rz -11.91 deg; joints [10.161, -29.249, 81.641, -91.066, 88.675, 141.53]
  MoveL 1561 to (-195.21, 422.52, -13.48) mm, rotated rx -180 ry 0 rz -11.91 deg; joints [10.169, -29.248, 81.638, -91.06, 88.68, 141.528]
  MoveL 1562 to (-194.97, 422.52, -13.48) mm, rotated rx 180 ry 0 rz -11.91 deg; joints [10.177, -29.246, 81.633, -91.054, 88.685, 141.526]
  Set speed (38.1 mm/s)
  MoveL 1563 to (-194.97, 421.25, -13.48) mm, rotated rx -180 ry 0 rz -11.91 deg; joints [10.185, -29.312, 81.778, -91.049, 88.691, 141.604]
  MoveL 1564 to (-195.61, 421.25, -13.48) mm, rotated rx -180 ry 0 rz -11.91 deg; joints [10.164, -29.318, 81.791, -91.066, 88.678, 141.611]
  Set speed (25.4 mm/s)
  MoveL 1565 to (-195.61, 421.25, -15.84) mm, rotated rx -180 ry 0 rz -11.91 deg; joints [10.165, -29.207, 81.766, -91.068, 88.68, 141.697]
  MoveL 1566 to (-195.61, 421.89, -16.47) mm, rotated rx 180 ry 0 rz -11.91 deg; joints [10.161, -29.144, 81.686, -91.07, 88.678, 141.681]
  Set speed (38.1 mm/s)
  MoveL 1567 to (-194.97, 422.52, -16.48) mm, rotated rx 180 ry 0 rz -11.91 deg; joints [10.178, -29.104, 81.601, -91.056, 88.687, 141.634]
  Set speed (76.2 mm/s)
  MoveL 1568 to (213.41, 422.52, -16.48) mm, rotated rx -180 ry 0 rz -11.91 deg; joints [22.901, -22.259, 66.588, -81.918, 97.625, 134.038]
  MoveL 1569 to (213.89, 422.53, -16.48) mm, rotated rx -180 ry 0 rz -11.91 deg; joints [22.915, -22.246, 66.56, -81.91, 97.637, 134.025]
  MoveL 1570 to (214.13, 422.55, -16.47) mm, rotated rx 180 ry 0 rz -11.91 deg; joints [22.921, -22.238, 66.543, -81.907, 97.643, 134.017]
  MoveL 1571 to (214.37, 422.59, -16.47) mm, rotated rx -180 ry 0 rz -11.91 deg; joints [22.928, -22.23, 66.524, -81.904, 97.649, 134.007]
  MoveL 1572 to (214.61, 422.65, -16.47) mm, rotated rx -180 ry 0 rz -11.91 deg; joints [22.934, -22.219, 66.503, -81.901, 97.655, 133.996]
  MoveL 1573 to (214.85, 422.74, -16.48) mm, rotated rx -180 ry 0 rz -11.91 deg; joints [22.94, -22.208, 66.478, -81.898, 97.661, 133.984]
  MoveL 1574 to (215.09, 422.84, -16.47) mm, rotated rx -180 ry 0 rz -11.91 deg; joints [22.946, -22.195, 66.451, -81.896, 97.667, 133.97]
  MoveL 1575 to (215.34, 422.97, -16.47) mm, rotated rx 180 ry 0 rz -11.91 deg; joints [22.951, -22.181, 66.42, -81.895, 97.673, 133.954]
  MoveL 1576 to (215.58, 423.13, -16.47) mm, rotated rx -180 ry 0 rz -11.91 deg; joints [22.956, -22.165, 66.385, -81.893, 97.679, 133.936]
  MoveL 1577 to (215.82, 423.33, -16.47) mm, rotated rx -180 ry 0 rz -11.91 deg; joints [22.96, -22.146, 66.346, -81.893, 97.685, 133.916]
  MoveL 1578 to (215.96, 423.46, -16.48) mm, rotated rx -180 ry 0 rz -11.91 deg; joints [22.963, -22.134, 66.32, -81.893, 97.689, 133.902]
  MoveL 1579 to (216.09, 423.6, -16.47) mm, rotated rx -180 ry 0 rz -11.91 deg; joints [22.965, -22.122, 66.295, -81.893, 97.692, 133.889]
  MoveL 1580 to (216.2, 423.73, -16.48) mm, rotated rx 180 ry 0 rz -11.91 deg; joints [22.966, -22.111, 66.271, -81.894, 97.695, 133.877]
  MoveL 1581 to (216.3, 423.87, -16.48) mm, rotated rx 180 ry 0 rz -11.91 deg; joints [22.968, -22.1, 66.247, -81.895, 97.698, 133.864]
  MoveL 1582 to (216.39, 424.01, -16.48) mm, rotated rx -180 ry 0 rz -11.91 deg; joints [22.969, -22.089, 66.224, -81.896, 97.7, 133.852]
  MoveL 1583 to (216.47, 424.15, -16.48) mm, rotated rx 180 ry 0 rz -11.91 deg; joints [22.969, -22.078, 66.201, -81.897, 97.702, 133.84]
  MoveL 1584 to (216.69, 424.27, -16.48) mm, rotated rx 180 ry 0 rz -11.91 deg; joints [22.974, -22.065, 66.172, -81.896, 97.708, 133.825]
  MoveL 1585 to (219.83, 424.27, -16.48) mm, rotated rx 180 ry 0 rz -11.91 deg; joints [23.065, -21.982, 65.995, -81.844, 97.786, 133.74]
  MoveL 1586 to (220.05, 424.15, -16.48) mm, rotated rx -180 ry 0 rz -11.91 deg; joints [23.073, -21.984, 65.998, -81.838, 97.791, 133.742]
  MoveL 1587 to (220.05, 53.41, -16.48) mm, rotated rx 180 ry 0 rz -11.91 deg; joints [28.67, -39.062, 103.469, -74.55, 96.833, 154.525]
  MoveL 1588 to (219.83, 53.17, -16.48) mm, rotated rx 180 ry 0 rz -11.91 deg; joints [28.667, -39.075, 103.498, -74.551, 96.827, 154.541]
  MoveL 1589 to (-196.42, 53.17, -16.48) mm, rotated rx -180 ry 0 rz -11.91 deg; joints [12.924, -44.371, 116.688, -88.822, 89.957, 161.451]
  MoveL 1590 to (-196.42, 53.41, -16.47) mm, rotated rx -180 ry 0 rz -11.91 deg; joints [12.921, -44.364, 116.668, -88.824, 89.956, 161.44]
  MoveL 1591 to (-196.42, 422.66, -16.48) mm, rotated rx -180 ry 0 rz -11.91 deg; joints [10.129, -29.111, 81.615, -91.094, 88.658, 141.643]
  MoveL 1592 to (-196.42, 422.81, -16.48) mm, rotated rx 180 ry 0 rz -11.91 deg; joints [10.129, -29.103, 81.598, -91.095, 88.657, 141.634]
  MoveL 1593 to (-196.18, 422.71, -16.48) mm, rotated rx -180 ry 0 rz -11.91 deg; joints [10.137, -29.106, 81.604, -91.088, 88.663, 141.637]
  MoveL 1594 to (-195.93, 422.63, -16.48) mm, rotated rx 180 ry 0 rz -11.91 deg; joints [10.146, -29.107, 81.608, -91.081, 88.668, 141.639]
  MoveL 1595 to (-195.69, 422.58, -16.47) mm, rotated rx -180 ry 0 rz -11.91 deg; joints [10.154, -29.108, 81.609, -91.075, 88.673, 141.64]
  MoveL 1596 to (-195.45, 422.54, -16.48) mm, rotated rx 180 ry 0 rz -11.91 deg; joints [10.162, -29.108, 81.609, -91.068, 88.678, 141.639]
  MoveL 1597 to (-195.21, 422.52, -16.48) mm, rotated rx -180 ry 0 rz -11.91 deg; joints [10.17, -29.107, 81.606, -91.062, 88.683, 141.637]
  MoveL 1598 to (-194.97, 422.52, -16.48) mm, rotated rx 180 ry 0 rz -11.91 deg; joints [10.178, -29.104, 81.601, -91.056, 88.687, 141.634]
  MoveL 1599 to (-164.9, 422.52, -17.52) mm, rotated rx 180 ry 0 rz -11.91 deg; joints [11.168, -28.765, 80.938, -90.266, 89.289, 141.304]
  MoveL 1600 to (213.41, 422.52, -17.52) mm, rotated rx -180 ry 0 rz -11.91 deg; joints [22.901, -22.212, 66.575, -81.914, 97.62, 134.072]
  MoveL 1601 to (213.89, 422.53, -17.52) mm, rotated rx -180 ry 0 rz -11.91 deg; joints [22.915, -22.199, 66.547, -81.906, 97.632, 134.059]
  MoveL 1602 to (214.13, 422.55, -17.53) mm, rotated rx -180 ry 0 rz -11.91 deg; joints [22.922, -22.192, 66.53, -81.902, 97.638, 134.051]
  MoveL 1603 to (214.37, 422.59, -17.53) mm, rotated rx 180 ry 0 rz -11.91 deg; joints [22.928, -22.183, 66.511, -81.899, 97.644, 134.041]
  MoveL 1604 to (214.61, 422.65, -17.52) mm, rotated rx -180 ry 0 rz -11.91 deg; joints [22.934, -22.173, 66.49, -81.896, 97.65, 134.03]
  MoveL 1605 to (214.85, 422.74, -17.53) mm, rotated rx 180 ry 0 rz -11.91 deg; joints [22.94, -22.161, 66.465, -81.894, 97.656, 134.018]
  MoveL 1606 to (215.09, 422.84, -17.53) mm, rotated rx -180 ry 0 rz -11.91 deg; joints [22.946, -22.148, 66.438, -81.891, 97.662, 134.004]
  MoveL 1607 to (215.34, 422.97, -17.52) mm, rotated rx -180 ry 0 rz -11.91 deg; joints [22.951, -22.134, 66.407, -81.89, 97.668, 133.988]
  MoveL 1608 to (215.58, 423.13, -17.53) mm, rotated rx -180 ry 0 rz -11.91 deg; joints [22.956, -22.118, 66.372, -81.889, 97.674, 133.97]
  MoveL 1609 to (215.82, 423.33, -17.53) mm, rotated rx -180 ry 0 rz -11.91 deg; joints [22.961, -22.099, 66.333, -81.888, 97.681, 133.95]
  MoveL 1610 to (215.96, 423.46, -17.52) mm, rotated rx 180 ry 0 rz -11.91 deg; joints [22.963, -22.087, 66.307, -81.888, 97.684, 133.936]
  MoveL 1611 to (216.09, 423.6, -17.53) mm, rotated rx 180 ry 0 rz -11.91 deg; joints [22.965, -22.075, 66.282, -81.889, 97.688, 133.923]
  MoveL 1612 to (216.2, 423.73, -17.53) mm, rotated rx -180 ry 0 rz -11.91 deg; joints [22.967, -22.064, 66.258, -81.889, 97.691, 133.91]
  MoveL 1613 to (216.3, 423.87, -17.52) mm, rotated rx -180 ry 0 rz -11.91 deg; joints [22.968, -22.053, 66.234, -81.89, 97.693, 133.898]
  MoveL 1614 to (216.39, 424.01, -17.53) mm, rotated rx -180 ry 0 rz -11.91 deg; joints [22.969, -22.042, 66.211, -81.891, 97.696, 133.886]
  MoveL 1615 to (216.47, 424.15, -17.53) mm, rotated rx -180 ry 0 rz -11.91 deg; joints [22.97, -22.031, 66.188, -81.892, 97.698, 133.874]
  MoveL 1616 to (216.69, 424.27, -17.52) mm, rotated rx -180 ry 0 rz -11.91 deg; joints [22.975, -22.018, 66.159, -81.891, 97.703, 133.859]
  MoveL 1617 to (219.83, 424.27, -17.52) mm, rotated rx -180 ry 0 rz -11.91 deg; joints [23.065, -21.935, 65.982, -81.84, 97.781, 133.773]
  MoveL 1618 to (220.05, 424.15, -17.53) mm, rotated rx 180 ry 0 rz -11.91 deg; joints [23.073, -21.937, 65.985, -81.834, 97.787, 133.776]
  MoveL 1619 to (220.05, 53.41, -17.52) mm, rotated rx -180 ry 0 rz -11.91 deg; joints [28.671, -39.005, 103.458, -74.544, 96.821, 154.57]
  MoveL 1620 to (219.83, 53.17, -17.53) mm, rotated rx 180 ry 0 rz -11.91 deg; joints [28.667, -39.018, 103.487, -74.545, 96.815, 154.586]
  MoveL 1621 to (-195.15, 53.17, -17.52) mm, rotated rx -180 ry 0 rz -11.91 deg; joints [12.977, -44.297, 116.652, -88.772, 89.972, 161.49]
  MoveL 1622 to (-195.65, 53.17, -17.53) mm, rotated rx -180 ry 0 rz -11.91 deg; joints [12.956, -44.301, 116.662, -88.791, 89.966, 161.496]
  MoveL 1623 to (-195.81, 53.41, -17.52) mm, rotated rx -180 ry 0 rz -11.91 deg; joints [12.947, -44.295, 116.646, -88.8, 89.963, 161.486]
  MoveL 1624 to (-195.81, 422.38, -17.53) mm, rotated rx 180 ry 0 rz -11.91 deg; joints [10.151, -29.07, 81.623, -91.078, 88.672, 141.691]
  MoveL 1625 to (-195.65, 422.57, -17.53) mm, rotated rx -180 ry 0 rz -11.91 deg; joints [10.156, -29.059, 81.598, -91.074, 88.675, 141.678]
  MoveL 1626 to (-195.48, 422.55, -17.53) mm, rotated rx 180 ry 0 rz -11.91 deg; joints [10.161, -29.058, 81.597, -91.07, 88.678, 141.677]
  MoveL 1627 to (-195.32, 422.53, -17.52) mm, rotated rx -180 ry 0 rz -11.91 deg; joints [10.167, -29.058, 81.596, -91.065, 88.681, 141.676]
  MoveL 1628 to (-195.15, 422.52, -17.53) mm, rotated rx -180 ry 0 rz -11.91 deg; joints [10.172, -29.057, 81.593, -91.061, 88.685, 141.675]
  MoveL 1629 to (-194.97, 422.52, -17.53) mm, rotated rx -180 ry 0 rz -11.91 deg; joints [10.178, -29.055, 81.589, -91.056, 88.688, 141.672]
  MoveL 1630 to (-164.9, 422.52, -17.52) mm, rotated rx 180 ry 0 rz -11.91 deg; joints [11.168, -28.765, 80.938, -90.266, 89.289, 141.304]
  Set speed (38.1 mm/s)
  MoveL 1631 to (-164.28, 421.77, -17.53) mm, rotated rx 180 ry 0 rz -11.91 deg; joints [11.194, -28.798, 81.009, -90.246, 89.304, 141.343]
  MoveL 1632 to (-164.81, 418.84, -17.52) mm, rotated rx -180 ry 0 rz -11.91 deg; joints [11.195, -28.957, 81.357, -90.247, 89.306, 141.531]
  MoveL 1633 to (-164.93, 418.21, -16.89) mm, rotated rx -180 ry 0 rz -11.91 deg; joints [11.195, -29.021, 81.438, -90.247, 89.306, 141.548]
  Set speed (100.0 mm/s)
  MoveL 1634 to (-164.93, 418.21, 24.53) mm, rotated rx 180 ry 0 rz -11.91 deg; joints [11.186, -30.941, 81.818, -90.236, 89.294, 140.008]
  MoveL 1635 to (-164.87, 434.05, 24.53) mm, rotated rx 180 ry 0 rz -11.91 deg; joints [11.085, -30.085, 79.996, -90.301, 89.225, 139.043]
  MoveL 1636 to (-164.87, 434.05, -6.52) mm, rotated rx -180 ry 0 rz -11.91 deg; joints [11.092, -28.664, 79.722, -90.311, 89.236, 140.189]
  Set speed (25.4 mm/s)
  MoveL 1637 to (-164.87, 434.05, -9.84) mm, rotated rx 180 ry 0 rz -11.91 deg; joints [11.093, -28.51, 79.688, -90.312, 89.237, 140.309]
  MoveL 1638 to (-164.72, 433.43, -10.48) mm, rotated rx -180 ry 0 rz -11.91 deg; joints [11.102, -28.512, 79.75, -90.306, 89.243, 140.369]
  Set speed (38.1 mm/s)
  MoveL 1639 to (-164.28, 431.48, -10.48) mm, rotated rx 180 ry 0 rz -11.91 deg; joints [11.129, -28.612, 79.966, -90.287, 89.26, 140.485]
  MoveL 1640 to (-164.9, 430.7, -10.48) mm, rotated rx 180 ry 0 rz -11.91 deg; joints [11.113, -28.66, 80.07, -90.299, 89.251, 140.541]
  Set speed (76.2 mm/s)
  MoveL 1641 to (-194.97, 430.7, -10.48) mm, rotated rx -180 ry 0 rz -11.91 deg; joints [10.128, -28.954, 80.726, -91.078, 88.643, 140.91]
  MoveL 1642 to (-202.2, 430.7, -10.48) mm, rotated rx -180 ry 0 rz -11.91 deg; joints [9.89, -29.021, 80.874, -91.267, 88.498, 140.995]
  MoveL 1643 to (-203.17, 430.7, -10.48) mm, rotated rx -180 ry 0 rz -11.91 deg; joints [9.858, -29.029, 80.894, -91.293, 88.478, 141.006]
  MoveL 1644 to (-203.41, 430.69, -10.47) mm, rotated rx -180 ry 0 rz -11.91 deg; joints [9.851, -29.032, 80.901, -91.299, 88.474, 141.01]
  MoveL 1645 to (-203.65, 430.65, -10.48) mm, rotated rx -180 ry 0 rz -11.91 deg; joints [9.843, -29.037, 80.91, -91.305, 88.469, 141.015]
  MoveL 1646 to (-203.89, 430.6, -10.48) mm, rotated rx 180 ry 0 rz -11.91 deg; joints [9.835, -29.042, 80.921, -91.311, 88.464, 141.021]
  MoveL 1647 to (-204.13, 430.52, -10.47) mm, rotated rx -180 ry 0 rz -11.91 deg; joints [9.828, -29.048, 80.934, -91.317, 88.46, 141.029]
  MoveL 1648 to (-204.42, 430.43, -10.48) mm, rotated rx -180 ry 0 rz -11.91 deg; joints [9.819, -29.055, 80.951, -91.325, 88.455, 141.038]
  MoveL 1649 to (-204.57, 430.37, -10.47) mm, rotated rx -180 ry 0 rz -11.91 deg; joints [9.814, -29.06, 80.96, -91.328, 88.452, 141.043]
  MoveL 1650 to (-204.72, 430.31, -10.47) mm, rotated rx 180 ry 0 rz -11.91 deg; joints [9.81, -29.064, 80.971, -91.332, 88.449, 141.049]
  MoveL 1651 to (-204.86, 430.23, -10.48) mm, rotated rx 180 ry 0 rz -11.91 deg; joints [9.805, -29.07, 80.982, -91.336, 88.447, 141.055]
  MoveL 1652 to (-205.01, 430.15, -10.47) mm, rotated rx -180 ry 0 rz -11.91 deg; joints [9.801, -29.075, 80.995, -91.339, 88.444, 141.062]
  MoveL 1653 to (-205.16, 430.05, -10.48) mm, rotated rx -180 ry 0 rz -11.91 deg; joints [9.797, -29.082, 81.009, -91.343, 88.442, 141.07]
  MoveL 1654 to (-205.3, 429.94, -10.48) mm, rotated rx -180 ry 0 rz -11.91 deg; joints [9.792, -29.089, 81.024, -91.346, 88.439, 141.078]
  MoveL 1655 to (-205.53, 429.75, -10.48) mm, rotated rx 180 ry 0 rz -11.91 deg; joints [9.786, -29.101, 81.051, -91.352, 88.436, 141.093]
  MoveL 1656 to (-205.75, 429.52, -10.48) mm, rotated rx 180 ry 0 rz -11.91 deg; joints [9.78, -29.115, 81.082, -91.357, 88.433, 141.11]
  MoveL 1657 to (-205.92, 429.3, -10.48) mm, rotated rx -180 ry 0 rz -11.91 deg; joints [9.776, -29.128, 81.11, -91.361, 88.43, 141.125]
  MoveL 1658 to (-206.06, 429.09, -10.48) mm, rotated rx -180 ry 0 rz -11.91 deg; joints [9.772, -29.141, 81.137, -91.364, 88.428, 141.14]
  MoveL 1659 to (-206.14, 428.96, -10.48) mm, rotated rx -180 ry 0 rz -11.91 deg; joints [9.771, -29.149, 81.155, -91.366, 88.428, 141.149]
  MoveL 1660 to (-206.21, 428.82, -10.48) mm, rotated rx -180 ry 0 rz -11.91 deg; joints [9.769, -29.156, 81.171, -91.367, 88.427, 141.158]
  MoveL 1661 to (-206.27, 428.69, -10.48) mm, rotated rx -180 ry 0 rz -11.91 deg; joints [9.768, -29.164, 81.188, -91.368, 88.426, 141.167]
  MoveL 1662 to (-206.32, 428.55, -10.48) mm, rotated rx -180 ry 0 rz -11.91 deg; joints [9.767, -29.172, 81.205, -91.369, 88.426, 141.176]
  MoveL 1663 to (-206.37, 428.42, -10.47) mm, rotated rx -180 ry 0 rz -11.91 deg; joints [9.766, -29.179, 81.221, -91.37, 88.426, 141.185]
  MoveL 1664 to (-206.41, 428.28, -10.47) mm, rotated rx -180 ry 0 rz -11.91 deg; joints [9.765, -29.187, 81.237, -91.371, 88.426, 141.194]
  MoveL 1665 to (-206.47, 428.01, -10.47) mm, rotated rx -180 ry 0 rz -11.91 deg; joints [9.765, -29.202, 81.27, -91.372, 88.426, 141.211]
  MoveL 1666 to (-206.5, 427.77, -10.48) mm, rotated rx 180 ry 0 rz -11.91 deg; joints [9.765, -29.215, 81.298, -91.372, 88.426, 141.227]
  MoveL 1667 to (-206.52, 427.53, -10.47) mm, rotated rx -180 ry 0 rz -11.91 deg; joints [9.766, -29.228, 81.326, -91.372, 88.427, 141.242]
  MoveL 1668 to (-206.52, 427.04, -10.48) mm, rotated rx 180 ry 0 rz -11.91 deg; joints [9.769, -29.253, 81.381, -91.37, 88.429, 141.272]
  MoveL 1669 to (-206.52, 50.21, -10.47) mm, rotated rx 180 ry 0 rz -11.91 deg; joints [12.529, -44.912, 117.182, -89.198, 89.838, 161.403]
  MoveL 1670 to (-206.51, 49.73, -10.47) mm, rotated rx -180 ry 0 rz -11.91 deg; joints [12.534, -44.927, 117.221, -89.193, 89.839, 161.427]
  MoveL 1671 to (-206.48, 49.48, -10.47) mm, rotated rx -180 ry 0 rz -11.91 deg; joints [12.538, -44.935, 117.241, -89.189, 89.84, 161.438]
  MoveL 1672 to (-206.43, 49.24, -10.47) mm, rotated rx -180 ry 0 rz -11.91 deg; joints [12.542, -44.943, 117.26, -89.185, 89.841, 161.45]
  MoveL 1673 to (-206.37, 49.02, -10.48) mm, rotated rx -180 ry 0 rz -11.91 deg; joints [12.547, -44.95, 117.277, -89.181, 89.842, 161.46]
  MoveL 1674 to (-206.28, 48.8, -10.48) mm, rotated rx -180 ry 0 rz -11.91 deg; joints [12.553, -44.957, 117.293, -89.176, 89.844, 161.47]
  MoveL 1675 to (-206.18, 48.57, -10.48) mm, rotated rx 180 ry 0 rz -11.91 deg; joints [12.559, -44.963, 117.31, -89.17, 89.846, 161.48]
  MoveL 1676 to (-206.06, 48.35, -10.48) mm, rotated rx 180 ry 0 rz -11.91 deg; joints [12.566, -44.97, 117.326, -89.163, 89.848, 161.489]
  MoveL 1677 to (-205.98, 48.22, -10.47) mm, rotated rx -180 ry 0 rz -11.91 deg; joints [12.571, -44.973, 117.335, -89.158, 89.849, 161.495]
  MoveL 1678 to (-205.88, 48.09, -10.48) mm, rotated rx 180 ry 0 rz -11.91 deg; joints [12.576, -44.977, 117.344, -89.153, 89.851, 161.5]
  MoveL 1679 to (-205.78, 47.96, -10.48) mm, rotated rx 180 ry 0 rz -11.91 deg; joints [12.582, -44.981, 117.353, -89.148, 89.852, 161.505]
  MoveL 1680 to (-205.66, 47.83, -10.48) mm, rotated rx -180 ry 0 rz -11.91 deg; joints [12.588, -44.984, 117.361, -89.142, 89.854, 161.51]
  MoveL 1681 to (-205.51, 47.67, -10.48) mm, rotated rx 180 ry 0 rz -11.91 deg; joints [12.596, -44.988, 117.371, -89.135, 89.856, 161.516]
  MoveL 1682 to (-205.35, 47.54, -10.48) mm, rotated rx -180 ry 0 rz -11.91 deg; joints [12.604, -44.992, 117.38, -89.127, 89.859, 161.521]
  MoveL 1683 to (-205.19, 47.42, -10.47) mm, rotated rx -180 ry 0 rz -11.91 deg; joints [12.611, -44.995, 117.387, -89.12, 89.861, 161.525]
  MoveL 1684 to (-205.03, 47.31, -10.48) mm, rotated rx -180 ry 0 rz -11.91 deg; joints [12.619, -44.997, 117.392, -89.113, 89.863, 161.529]
  MoveL 1685 to (-204.81, 47.18, -10.48) mm, rotated rx 180 ry 0 rz -11.91 deg; joints [12.629, -45, 117.399, -89.103, 89.866, 161.532]
  MoveL 1686 to (-204.58, 47.08, -10.47) mm, rotated rx 180 ry 0 rz -11.91 deg; joints [12.64, -45.001, 117.403, -89.093, 89.869, 161.535]
  MoveL 1687 to (-204.36, 46.99, -10.47) mm, rotated rx -180 ry 0 rz -11.91 deg; joints [12.65, -45.003, 117.406, -89.083, 89.872, 161.537]
  MoveL 1688 to (-204.13, 46.92, -10.48) mm, rotated rx -180 ry 0 rz -11.91 deg; joints [12.66, -45.003, 117.407, -89.073, 89.875, 161.538]
  MoveL 1689 to (-203.89, 46.87, -10.47) mm, rotated rx 180 ry 0 rz -11.91 deg; joints [12.671, -45.003, 117.407, -89.063, 89.879, 161.537]
  MoveL 1690 to (-203.65, 46.84, -10.47) mm, rotated rx 180 ry 0 rz -11.91 deg; joints [12.681, -45.003, 117.405, -89.053, 89.882, 161.536]
  MoveL 1691 to (-203.41, 46.83, -10.48) mm, rotated rx -180 ry 0 rz -11.91 deg; joints [12.691, -45.002, 117.402, -89.044, 89.885, 161.534]
  MoveL 1692 to (-203.17, 46.83, -10.47) mm, rotated rx -180 ry 0 rz -11.91 deg; joints [12.701, -45, 117.398, -89.034, 89.888, 161.531]
  MoveL 1693 to (222.09, 46.82, -10.48) mm, rotated rx 180 ry 0 rz -11.91 deg; joints [28.858, -39.583, 103.974, -74.38, 96.915, 154.532]
  MoveL 1694 to (223.29, 46.83, -10.48) mm, rotated rx -180 ry 0 rz -11.91 deg; joints [28.898, -39.561, 103.92, -74.346, 96.941, 154.506]
  MoveL 1695 to (223.53, 46.84, -10.48) mm, rotated rx 180 ry 0 rz -11.91 deg; joints [28.906, -39.555, 103.908, -74.34, 96.946, 154.5]
  MoveL 1696 to (223.77, 46.87, -10.47) mm, rotated rx 180 ry 0 rz -11.91 deg; joints [28.914, -39.55, 103.895, -74.334, 96.951, 154.494]
  MoveL 1697 to (224.01, 46.92, -10.47) mm, rotated rx -180 ry 0 rz -11.91 deg; joints [28.921, -39.543, 103.88, -74.328, 96.956, 154.486]
  MoveL 1698 to (224.24, 46.99, -10.47) mm, rotated rx -180 ry 0 rz -11.91 deg; joints [28.927, -39.537, 103.864, -74.324, 96.961, 154.478]
  MoveL 1699 to (224.46, 47.08, -10.48) mm, rotated rx 180 ry 0 rz -11.91 deg; joints [28.933, -39.529, 103.847, -74.319, 96.967, 154.47]
  MoveL 1700 to (224.69, 47.18, -10.48) mm, rotated rx 180 ry 0 rz -11.91 deg; joints [28.939, -39.521, 103.828, -74.315, 96.972, 154.46]
  MoveL 1701 to (224.92, 47.31, -10.48) mm, rotated rx 180 ry 0 rz -11.91 deg; joints [28.944, -39.513, 103.808, -74.312, 96.977, 154.449]
  MoveL 1702 to (225.07, 47.42, -10.47) mm, rotated rx -180 ry 0 rz -11.91 deg; joints [28.947, -39.506, 103.792, -74.31, 96.981, 154.441]
  MoveL 1703 to (225.23, 47.54, -10.47) mm, rotated rx -180 ry 0 rz -11.91 deg; joints [28.95, -39.499, 103.775, -74.308, 96.985, 154.432]
  MoveL 1704 to (225.39, 47.67, -10.48) mm, rotated rx 180 ry 0 rz -11.91 deg; joints [28.953, -39.491, 103.757, -74.307, 96.989, 154.422]
  MoveL 1705 to (225.55, 47.83, -10.47) mm, rotated rx 180 ry 0 rz -11.91 deg; joints [28.955, -39.482, 103.737, -74.306, 96.993, 154.411]
  MoveL 1706 to (225.66, 47.96, -10.47) mm, rotated rx 180 ry 0 rz -11.91 deg; joints [28.957, -39.475, 103.721, -74.306, 96.996, 154.403]
  MoveL 1707 to (225.77, 48.09, -10.48) mm, rotated rx -180 ry 0 rz -11.91 deg; joints [28.958, -39.469, 103.706, -74.306, 96.999, 154.395]
  MoveL 1708 to (225.86, 48.22, -10.48) mm, rotated rx 180 ry 0 rz -11.91 deg; joints [28.959, -39.462, 103.691, -74.306, 97.001, 154.387]
  MoveL 1709 to (225.94, 48.35, -10.48) mm, rotated rx -180 ry 0 rz -11.91 deg; joints [28.959, -39.456, 103.677, -74.307, 97.004, 154.379]
  MoveL 1710 to (226.07, 48.57, -10.48) mm, rotated rx 180 ry 0 rz -11.91 deg; joints [28.959, -39.446, 103.653, -74.309, 97.007, 154.366]
  MoveL 1711 to (226.17, 48.8, -10.48) mm, rotated rx -180 ry 0 rz -11.91 deg; joints [28.958, -39.436, 103.631, -74.311, 97.01, 154.353]
  MoveL 1712 to (226.25, 49.02, -10.47) mm, rotated rx -180 ry 0 rz -11.91 deg; joints [28.957, -39.427, 103.609, -74.314, 97.013, 154.341]
  MoveL 1713 to (226.31, 49.24, -10.47) mm, rotated rx 180 ry 0 rz -11.91 deg; joints [28.955, -39.418, 103.588, -74.317, 97.015, 154.329]
  MoveL 1714 to (226.36, 49.48, -10.47) mm, rotated rx -180 ry 0 rz -11.91 deg; joints [28.952, -39.408, 103.566, -74.321, 97.018, 154.317]
  MoveL 1715 to (226.39, 49.73, -10.48) mm, rotated rx -180 ry 0 rz -11.91 deg; joints [28.948, -39.399, 103.545, -74.325, 97.019, 154.305]
  MoveL 1716 to (226.4, 50.21, -10.48) mm, rotated rx -180 ry 0 rz -11.91 deg; joints [28.94, -39.382, 103.505, -74.336, 97.022, 154.282]
  MoveL 1717 to (226.4, 427.53, -10.48) mm, rotated rx -180 ry 0 rz -11.91 deg; joints [23.212, -21.867, 65.255, -81.826, 97.98, 133.131]
  MoveL 1718 to (226.39, 427.77, -10.48) mm, rotated rx 180 ry 0 rz -11.91 deg; joints [23.208, -21.852, 65.223, -81.831, 97.98, 133.113]
  MoveL 1719 to (226.37, 428.01, -10.47) mm, rotated rx 180 ry 0 rz -11.91 deg; joints [23.205, -21.837, 65.192, -81.836, 97.979, 133.097]
  MoveL 1720 to (226.34, 428.16, -10.47) mm, rotated rx 180 ry 0 rz -11.91 deg; joints [23.202, -21.829, 65.174, -81.839, 97.979, 133.087]
  MoveL 1721 to (226.31, 428.3, -10.47) mm, rotated rx -180 ry 0 rz -11.91 deg; joints [23.199, -21.82, 65.157, -81.842, 97.978, 133.077]
  MoveL 1722 to (226.27, 428.45, -10.47) mm, rotated rx -180 ry 0 rz -11.91 deg; joints [23.196, -21.812, 65.139, -81.845, 97.977, 133.068]
  MoveL 1723 to (226.22, 428.59, -10.48) mm, rotated rx 180 ry 0 rz -11.91 deg; joints [23.193, -21.804, 65.122, -81.849, 97.976, 133.059]
  MoveL 1724 to (226.16, 428.74, -10.48) mm, rotated rx 180 ry 0 rz -11.91 deg; joints [23.19, -21.796, 65.106, -81.852, 97.975, 133.05]
  MoveL 1725 to (226.1, 428.89, -10.47) mm, rotated rx -180 ry 0 rz -11.91 deg; joints [23.186, -21.789, 65.09, -81.856, 97.974, 133.041]
  MoveL 1726 to (226.03, 429.03, -10.48) mm, rotated rx -180 ry 0 rz -11.91 deg; joints [23.182, -21.781, 65.075, -81.86, 97.972, 133.033]
  MoveL 1727 to (225.94, 429.18, -10.48) mm, rotated rx -180 ry 0 rz -11.91 deg; joints [23.178, -21.774, 65.06, -81.864, 97.97, 133.024]
  MoveL 1728 to (225.82, 429.37, -10.48) mm, rotated rx 180 ry 0 rz -11.91 deg; joints [23.172, -21.765, 65.041, -81.87, 97.967, 133.014]
  MoveL 1729 to (225.67, 429.56, -10.48) mm, rotated rx 180 ry 0 rz -11.91 deg; joints [23.165, -21.757, 65.024, -81.875, 97.964, 133.004]
  MoveL 1730 to (225.5, 429.75, -10.48) mm, rotated rx 180 ry 0 rz -11.91 deg; joints [23.158, -21.75, 65.008, -81.882, 97.959, 132.995]
  MoveL 1731 to (225.29, 429.94, -10.48) mm, rotated rx -180 ry 0 rz -11.91 deg; joints [23.15, -21.743, 64.994, -81.889, 97.954, 132.987]
  MoveL 1732 to (225.13, 430.07, -10.48) mm, rotated rx 180 ry 0 rz -11.91 deg; joints [23.144, -21.739, 64.986, -81.893, 97.951, 132.982]
  MoveL 1733 to (224.97, 430.18, -10.48) mm, rotated rx -180 ry 0 rz -11.91 deg; joints [23.138, -21.736, 64.98, -81.898, 97.947, 132.979]
  MoveL 1734 to (224.81, 430.28, -10.48) mm, rotated rx -180 ry 0 rz -11.91 deg; joints [23.132, -21.734, 64.976, -81.902, 97.943, 132.976]
  MoveL 1735 to (224.65, 430.37, -10.48) mm, rotated rx -180 ry 0 rz -11.91 deg; joints [23.126, -21.733, 64.974, -81.906, 97.939, 132.974]
  MoveL 1736 to (224.49, 430.44, -10.48) mm, rotated rx 180 ry 0 rz -11.91 deg; joints [23.121, -21.733, 64.973, -81.91, 97.935, 132.973]
  MoveL 1737 to (224.33, 430.51, -10.48) mm, rotated rx 180 ry 0 rz -11.91 deg; joints [23.115, -21.733, 64.973, -81.914, 97.931, 132.973]
  MoveL 1738 to (224.17, 430.56, -10.47) mm, rotated rx -180 ry 0 rz -11.91 deg; joints [23.11, -21.734, 64.975, -81.918, 97.927, 132.974]
  MoveL 1739 to (224.01, 430.6, -10.48) mm, rotated rx -180 ry 0 rz -11.91 deg; joints [23.105, -21.735, 64.978, -81.921, 97.923, 132.975]
  MoveL 1740 to (223.77, 430.66, -10.47) mm, rotated rx -180 ry 0 rz -11.91 deg; joints [23.098, -21.738, 64.985, -81.926, 97.917, 132.978]
  MoveL 1741 to (223.53, 430.69, -10.47) mm, rotated rx -180 ry 0 rz -11.91 deg; joints [23.09, -21.743, 64.995, -81.93, 97.911, 132.982]
  MoveL 1742 to (223.29, 430.7, -10.47) mm, rotated rx -180 ry 0 rz -11.91 deg; joints [23.083, -21.748, 65.007, -81.934, 97.905, 132.988]
  MoveL 1743 to (223.05, 430.7, -10.48) mm, rotated rx 180 ry 0 rz -11.91 deg; joints [23.076, -21.755, 65.021, -81.938, 97.899, 132.995]
  MoveL 1744 to (-164.9, 430.7, -10.48) mm, rotated rx 180 ry 0 rz -11.91 deg; joints [11.113, -28.66, 80.07, -90.299, 89.251, 140.541]
  Set speed (38.1 mm/s)
  MoveL 1745 to (-165.25, 431.87, -10.47) mm, rotated rx -180 ry 0 rz -11.91 deg; joints [11.094, -28.601, 79.943, -90.313, 89.239, 140.473]
  MoveL 1746 to (-164.27, 432.52, -10.48) mm, rotated rx -180 ry 0 rz -11.91 deg; joints [11.122, -28.556, 79.844, -90.291, 89.256, 140.419]
  Set speed (25.4 mm/s)
  MoveL 1747 to (-164.27, 432.52, -12.84) mm, rotated rx 180 ry 0 rz -11.91 deg; joints [11.123, -28.446, 79.819, -90.291, 89.257, 140.504]
  MoveL 1748 to (-164.27, 431.89, -13.48) mm, rotated rx -180 ry 0 rz -11.91 deg; joints [11.127, -28.45, 79.886, -90.289, 89.26, 140.567]
  Set speed (38.1 mm/s)
  MoveL 1749 to (-164.9, 431.25, -13.47) mm, rotated rx -180 ry 0 rz -11.91 deg; joints [11.111, -28.491, 79.975, -90.302, 89.25, 140.615]
  Set speed (76.2 mm/s)
  MoveL 1750 to (-194.97, 431.25, -13.48) mm, rotated rx 180 ry 0 rz -11.91 deg; joints [10.125, -28.785, 80.631, -91.082, 88.643, 140.985]
  MoveL 1751 to (-201.24, 431.25, -13.48) mm, rotated rx -180 ry 0 rz -11.91 deg; joints [9.919, -28.842, 80.76, -91.246, 88.517, 141.059]
  MoveL 1752 to (-201.48, 431.25, -13.48) mm, rotated rx -180 ry 0 rz -11.91 deg; joints [9.911, -28.845, 80.765, -91.252, 88.512, 141.062]
  MoveL 1753 to (-201.72, 431.23, -13.48) mm, rotated rx -180 ry 0 rz -11.91 deg; joints [9.904, -28.848, 80.772, -91.259, 88.508, 141.066]
  MoveL 1754 to (-201.96, 431.19, -13.47) mm, rotated rx -180 ry 0 rz -11.91 deg; joints [9.896, -28.852, 80.782, -91.265, 88.503, 141.071]
  MoveL 1755 to (-202.2, 431.13, -13.48) mm, rotated rx -180 ry 0 rz -11.91 deg; joints [9.888, -28.857, 80.793, -91.271, 88.498, 141.077]
  MoveL 1756 to (-204.13, 430.52, -13.47) mm, rotated rx -180 ry 0 rz -11.91 deg; joints [9.828, -28.907, 80.902, -91.32, 88.463, 141.138]
  MoveL 1757 to (-204.42, 430.43, -13.48) mm, rotated rx -180 ry 0 rz -11.91 deg; joints [9.819, -28.915, 80.919, -91.327, 88.457, 141.147]
  MoveL 1758 to (-204.57, 430.37, -13.48) mm, rotated rx -180 ry 0 rz -11.91 deg; joints [9.815, -28.919, 80.929, -91.331, 88.455, 141.152]
  MoveL 1759 to (-204.72, 430.31, -13.48) mm, rotated rx -180 ry 0 rz -11.91 deg; joints [9.81, -28.924, 80.939, -91.334, 88.452, 141.158]
  MoveL 1760 to (-204.86, 430.23, -13.47) mm, rotated rx -180 ry 0 rz -11.91 deg; joints [9.806, -28.929, 80.951, -91.338, 88.45, 141.164]
  MoveL 1761 to (-205.01, 430.15, -13.48) mm, rotated rx -180 ry 0 rz -11.91 deg; joints [9.802, -28.935, 80.963, -91.342, 88.447, 141.171]
  MoveL 1762 to (-205.16, 430.05, -13.48) mm, rotated rx -180 ry 0 rz -11.91 deg; joints [9.797, -28.941, 80.977, -91.345, 88.445, 141.179]
  MoveL 1763 to (-205.3, 429.94, -13.48) mm, rotated rx -180 ry 0 rz -11.91 deg; joints [9.793, -28.948, 80.992, -91.349, 88.442, 141.187]
  MoveL 1764 to (-205.53, 429.75, -13.48) mm, rotated rx -180 ry 0 rz -11.91 deg; joints [9.787, -28.961, 81.019, -91.354, 88.439, 141.202]
  MoveL 1765 to (-205.75, 429.52, -13.47) mm, rotated rx -180 ry 0 rz -11.91 deg; joints [9.781, -28.975, 81.051, -91.359, 88.436, 141.219]
  MoveL 1766 to (-205.92, 429.3, -13.48) mm, rotated rx -180 ry 0 rz -11.91 deg; joints [9.776, -28.988, 81.078, -91.363, 88.433, 141.234]
  MoveL 1767 to (-206.06, 429.09, -13.48) mm, rotated rx 180 ry 0 rz -11.91 deg; joints [9.773, -29, 81.106, -91.366, 88.431, 141.249]
  MoveL 1768 to (-206.14, 428.95, -13.48) mm, rotated rx -180 ry 0 rz -11.91 deg; joints [9.771, -29.008, 81.123, -91.368, 88.431, 141.258]
  MoveL 1769 to (-206.21, 428.82, -13.47) mm, rotated rx 180 ry 0 rz -11.91 deg; joints [9.77, -29.016, 81.14, -91.369, 88.43, 141.267]
  MoveL 1770 to (-206.27, 428.69, -13.48) mm, rotated rx -180 ry 0 rz -11.91 deg; joints [9.768, -29.023, 81.156, -91.371, 88.429, 141.276]
  MoveL 1771 to (-206.32, 428.55, -13.48) mm, rotated rx -180 ry 0 rz -11.91 deg; joints [9.767, -29.031, 81.173, -91.372, 88.429, 141.285]
  MoveL 1772 to (-206.37, 428.42, -13.48) mm, rotated rx -180 ry 0 rz -11.91 deg; joints [9.767, -29.039, 81.189, -91.373, 88.429, 141.294]
  MoveL 1773 to (-206.41, 428.28, -13.48) mm, rotated rx 180 ry 0 rz -11.91 deg; joints [9.766, -29.046, 81.206, -91.373, 88.429, 141.303]
  MoveL 1774 to (-206.47, 428.01, -13.47) mm, rotated rx -180 ry 0 rz -11.91 deg; joints [9.766, -29.061, 81.238, -91.374, 88.429, 141.32]
  MoveL 1775 to (-206.5, 427.77, -13.48) mm, rotated rx 180 ry 0 rz -11.91 deg; joints [9.766, -29.074, 81.266, -91.374, 88.429, 141.336]
  MoveL 1776 to (-206.52, 427.53, -13.48) mm, rotated rx 180 ry 0 rz -11.91 deg; joints [9.767, -29.087, 81.294, -91.374, 88.43, 141.351]
  MoveL 1777 to (-206.52, 427.04, -13.48) mm, rotated rx -180 ry 0 rz -11.91 deg; joints [9.769, -29.112, 81.35, -91.373, 88.432, 141.381]
  MoveL 1778 to (-206.52, 50.21, -13.48) mm, rotated rx 180 ry 0 rz -11.91 deg; joints [12.53, -44.726, 117.151, -89.197, 89.836, 161.558]
  MoveL 1779 to (-206.51, 49.73, -13.48) mm, rotated rx 180 ry 0 rz -11.91 deg; joints [12.535, -44.741, 117.19, -89.192, 89.837, 161.582]
  MoveL 1780 to (-206.48, 49.48, -13.48) mm, rotated rx 180 ry 0 rz -11.91 deg; joints [12.539, -44.749, 117.209, -89.189, 89.838, 161.593]
  MoveL 1781 to (-206.43, 49.24, -13.48) mm, rotated rx 180 ry 0 rz -11.91 deg; joints [12.543, -44.757, 117.228, -89.185, 89.839, 161.604]
  MoveL 1782 to (-206.37, 49.02, -13.47) mm, rotated rx -180 ry 0 rz -11.91 deg; joints [12.548, -44.764, 117.245, -89.18, 89.84, 161.615]
  MoveL 1783 to (-206.28, 48.8, -13.48) mm, rotated rx -180 ry 0 rz -11.91 deg; joints [12.553, -44.77, 117.262, -89.175, 89.842, 161.625]
  MoveL 1784 to (-206.18, 48.57, -13.47) mm, rotated rx 180 ry 0 rz -11.91 deg; joints [12.56, -44.777, 117.278, -89.169, 89.844, 161.634]
  MoveL 1785 to (-206.06, 48.35, -13.47) mm, rotated rx -180 ry 0 rz -11.91 deg; joints [12.567, -44.784, 117.294, -89.162, 89.846, 161.644]
  MoveL 1786 to (-205.98, 48.22, -13.48) mm, rotated rx 180 ry 0 rz -11.91 deg; joints [12.572, -44.787, 117.304, -89.158, 89.847, 161.65]
  MoveL 1787 to (-205.88, 48.09, -13.48) mm, rotated rx 180 ry 0 rz -11.91 deg; joints [12.577, -44.791, 117.313, -89.153, 89.849, 161.655]
  MoveL 1788 to (-205.78, 47.96, -13.48) mm, rotated rx 180 ry 0 rz -11.91 deg; joints [12.582, -44.794, 117.321, -89.148, 89.85, 161.66]
  MoveL 1789 to (-205.66, 47.83, -13.47) mm, rotated rx 180 ry 0 rz -11.91 deg; joints [12.588, -44.798, 117.33, -89.142, 89.852, 161.665]
  MoveL 1790 to (-205.51, 47.67, -13.48) mm, rotated rx -180 ry 0 rz -11.91 deg; joints [12.597, -44.802, 117.34, -89.134, 89.854, 161.671]
  MoveL 1791 to (-205.35, 47.54, -13.48) mm, rotated rx -180 ry 0 rz -11.91 deg; joints [12.604, -44.805, 117.348, -89.127, 89.857, 161.676]
  MoveL 1792 to (-205.19, 47.42, -13.48) mm, rotated rx -180 ry 0 rz -11.91 deg; joints [12.612, -44.808, 117.355, -89.119, 89.859, 161.68]
  MoveL 1793 to (-205.03, 47.31, -13.48) mm, rotated rx -180 ry 0 rz -11.91 deg; joints [12.62, -44.811, 117.361, -89.112, 89.861, 161.684]
  MoveL 1794 to (-204.81, 47.18, -13.48) mm, rotated rx -180 ry 0 rz -11.91 deg; joints [12.63, -44.813, 117.367, -89.102, 89.864, 161.687]
  MoveL 1795 to (-204.58, 47.08, -13.48) mm, rotated rx -180 ry 0 rz -11.91 deg; joints [12.641, -44.815, 117.372, -89.092, 89.867, 161.69]
  MoveL 1796 to (-204.36, 46.99, -13.48) mm, rotated rx -180 ry 0 rz -11.91 deg; joints [12.651, -44.816, 117.375, -89.082, 89.87, 161.692]
  MoveL 1797 to (-204.13, 46.92, -13.47) mm, rotated rx -180 ry 0 rz -11.91 deg; joints [12.661, -44.817, 117.376, -89.073, 89.873, 161.692]
  MoveL 1798 to (-203.89, 46.87, -13.48) mm, rotated rx -180 ry 0 rz -11.91 deg; joints [12.672, -44.817, 117.376, -89.063, 89.876, 161.692]
  MoveL 1799 to (-203.65, 46.84, -13.48) mm, rotated rx 180 ry 0 rz -11.91 deg; joints [12.682, -44.816, 117.374, -89.053, 89.88, 161.691]
  MoveL 1800 to (-203.41, 46.83, -13.47) mm, rotated rx -180 ry 0 rz -11.91 deg; joints [12.692, -44.815, 117.371, -89.043, 89.883, 161.689]
  MoveL 1801 to (-203.17, 46.83, -13.47) mm, rotated rx -180 ry 0 rz -11.91 deg; joints [12.702, -44.813, 117.366, -89.033, 89.886, 161.686]
  MoveL 1802 to (222.09, 46.83, -13.48) mm, rotated rx -180 ry 0 rz -11.91 deg; joints [28.859, -39.42, 103.944, -74.363, 96.88, 154.662]
  MoveL 1803 to (223.29, 46.83, -13.47) mm, rotated rx -180 ry 0 rz -11.91 deg; joints [28.9, -39.397, 103.89, -74.329, 96.905, 154.636]
  MoveL 1804 to (223.53, 46.84, -13.47) mm, rotated rx -180 ry 0 rz -11.91 deg; joints [28.907, -39.392, 103.878, -74.323, 96.91, 154.63]
  MoveL 1805 to (223.77, 46.87, -13.47) mm, rotated rx 180 ry 0 rz -11.91 deg; joints [28.915, -39.386, 103.865, -74.317, 96.916, 154.623]
  MoveL 1806 to (224.01, 46.92, -13.47) mm, rotated rx -180 ry 0 rz -11.91 deg; joints [28.922, -39.38, 103.85, -74.311, 96.921, 154.616]
  MoveL 1807 to (224.24, 46.99, -13.48) mm, rotated rx -180 ry 0 rz -11.91 deg; joints [28.928, -39.374, 103.834, -74.307, 96.926, 154.608]
  MoveL 1808 to (224.46, 47.08, -13.47) mm, rotated rx -180 ry 0 rz -11.91 deg; joints [28.934, -39.366, 103.817, -74.302, 96.931, 154.599]
  MoveL 1809 to (224.69, 47.18, -13.48) mm, rotated rx 180 ry 0 rz -11.91 deg; joints [28.94, -39.358, 103.799, -74.298, 96.936, 154.589]
  MoveL 1810 to (224.92, 47.31, -13.47) mm, rotated rx 180 ry 0 rz -11.91 deg; joints [28.945, -39.349, 103.778, -74.295, 96.942, 154.579]
  MoveL 1811 to (225.07, 47.42, -13.47) mm, rotated rx 180 ry 0 rz -11.91 deg; joints [28.949, -39.343, 103.762, -74.293, 96.945, 154.57]
  MoveL 1812 to (225.23, 47.54, -13.48) mm, rotated rx -180 ry 0 rz -11.91 deg; joints [28.952, -39.336, 103.745, -74.291, 96.949, 154.561]
  MoveL 1813 to (225.39, 47.67, -13.48) mm, rotated rx -180 ry 0 rz -11.91 deg; joints [28.954, -39.328, 103.727, -74.29, 96.953, 154.552]
  MoveL 1814 to (225.55, 47.83, -13.47) mm, rotated rx -180 ry 0 rz -11.91 deg; joints [28.957, -39.319, 103.707, -74.289, 96.957, 154.541]
  MoveL 1815 to (225.66, 47.96, -13.47) mm, rotated rx -180 ry 0 rz -11.91 deg; joints [28.958, -39.312, 103.691, -74.289, 96.96, 154.532]
  MoveL 1816 to (225.77, 48.09, -13.48) mm, rotated rx -180 ry 0 rz -11.91 deg; joints [28.959, -39.306, 103.676, -74.289, 96.963, 154.524]
  MoveL 1817 to (225.86, 48.22, -13.48) mm, rotated rx -180 ry 0 rz -11.91 deg; joints [28.96, -39.299, 103.662, -74.289, 96.966, 154.516]
  MoveL 1818 to (225.94, 48.35, -13.47) mm, rotated rx -180 ry 0 rz -11.91 deg; joints [28.96, -39.293, 103.647, -74.29, 96.968, 154.508]
  MoveL 1819 to (226.07, 48.57, -13.47) mm, rotated rx 180 ry 0 rz -11.91 deg; joints [28.96, -39.283, 103.624, -74.292, 96.972, 154.495]
  MoveL 1820 to (226.17, 48.8, -13.48) mm, rotated rx 180 ry 0 rz -11.91 deg; joints [28.959, -39.273, 103.601, -74.294, 96.975, 154.482]
  MoveL 1821 to (226.25, 49.02, -13.48) mm, rotated rx -180 ry 0 rz -11.91 deg; joints [28.958, -39.264, 103.579, -74.297, 96.978, 154.47]
  MoveL 1822 to (226.31, 49.24, -13.48) mm, rotated rx -180 ry 0 rz -11.91 deg; joints [28.956, -39.255, 103.558, -74.3, 96.98, 154.459]
  MoveL 1823 to (226.36, 49.48, -13.47) mm, rotated rx 180 ry 0 rz -11.91 deg; joints [28.953, -39.245, 103.536, -74.304, 96.982, 154.446]
  MoveL 1824 to (226.39, 49.73, -13.47) mm, rotated rx -180 ry 0 rz -11.91 deg; joints [28.95, -39.236, 103.515, -74.309, 96.984, 154.434]
  MoveL 1825 to (226.4, 50.21, -13.47) mm, rotated rx -180 ry 0 rz -11.91 deg; joints [28.941, -39.219, 103.475, -74.319, 96.986, 154.411]
  MoveL 1826 to (226.4, 428.01, -13.48) mm, rotated rx -180 ry 0 rz -11.91 deg; joints [23.206, -21.704, 65.154, -81.821, 97.967, 133.192]
  MoveL 1827 to (226.4, 428.23, -13.48) mm, rotated rx 180 ry 0 rz -11.91 deg; joints [23.204, -21.69, 65.125, -81.825, 97.967, 133.177]
  MoveL 1828 to (226.38, 428.44, -13.48) mm, rotated rx 180 ry 0 rz -11.91 deg; joints [23.201, -21.677, 65.097, -81.829, 97.967, 133.162]
  MoveL 1829 to (226.35, 428.65, -13.47) mm, rotated rx -180 ry 0 rz -11.91 deg; joints [23.197, -21.664, 65.07, -81.834, 97.967, 133.147]
  MoveL 1830 to (226.3, 428.87, -13.48) mm, rotated rx -180 ry 0 rz -11.91 deg; joints [23.193, -21.652, 65.044, -81.839, 97.966, 133.133]
  MoveL 1831 to (226.24, 429.08, -13.48) mm, rotated rx -180 ry 0 rz -11.91 deg; joints [23.189, -21.64, 65.019, -81.844, 97.964, 133.119]
  MoveL 1832 to (226.16, 429.3, -13.47) mm, rotated rx 180 ry 0 rz -11.91 deg; joints [23.184, -21.628, 64.994, -81.849, 97.963, 133.106]
  MoveL 1833 to (226.06, 429.51, -13.48) mm, rotated rx 180 ry 0 rz -11.91 deg; joints [23.178, -21.617, 64.971, -81.854, 97.96, 133.093]
  MoveL 1834 to (225.94, 429.73, -13.47) mm, rotated rx -180 ry 0 rz -11.91 deg; joints [23.172, -21.606, 64.949, -81.86, 97.958, 133.081]
  MoveL 1835 to (225.8, 429.94, -13.48) mm, rotated rx -180 ry 0 rz -11.91 deg; joints [23.165, -21.596, 64.928, -81.867, 97.954, 133.069]
  MoveL 1836 to (225.6, 430.19, -13.47) mm, rotated rx 180 ry 0 rz -11.91 deg; joints [23.157, -21.586, 64.906, -81.874, 97.95, 133.057]
  MoveL 1837 to (225.35, 430.44, -13.47) mm, rotated rx -180 ry 0 rz -11.91 deg; joints [23.146, -21.577, 64.887, -81.883, 97.944, 133.046]
  MoveL 1838 to (225.13, 430.62, -13.48) mm, rotated rx -180 ry 0 rz -11.91 deg; joints [23.138, -21.571, 64.875, -81.89, 97.938, 133.039]
  MoveL 1839 to (224.91, 430.77, -13.47) mm, rotated rx -180 ry 0 rz -11.91 deg; joints [23.129, -21.567, 64.867, -81.896, 97.933, 133.034]
  MoveL 1840 to (224.68, 430.9, -13.47) mm, rotated rx 180 ry 0 rz -11.91 deg; joints [23.122, -21.565, 64.863, -81.902, 97.928, 133.031]
  MoveL 1841 to (224.46, 431, -13.48) mm, rotated rx 180 ry 0 rz -11.91 deg; joints [23.114, -21.565, 64.862, -81.907, 97.922, 133.03]
  MoveL 1842 to (224.24, 431.09, -13.47) mm, rotated rx 180 ry 0 rz -11.91 deg; joints [23.106, -21.565, 64.863, -81.912, 97.917, 133.03]
  MoveL 1843 to (224.01, 431.15, -13.48) mm, rotated rx -180 ry 0 rz -11.91 deg; joints [23.099, -21.567, 64.867, -81.917, 97.911, 133.031]
  MoveL 1844 to (223.77, 431.21, -13.47) mm, rotated rx 180 ry 0 rz -11.91 deg; joints [23.092, -21.57, 64.874, -81.922, 97.905, 133.034]
  MoveL 1845 to (223.53, 431.24, -13.48) mm, rotated rx -180 ry 0 rz -11.91 deg; joints [23.084, -21.575, 64.884, -81.926, 97.899, 133.039]
  MoveL 1846 to (223.29, 431.25, -13.47) mm, rotated rx 180 ry 0 rz -11.91 deg; joints [23.077, -21.58, 64.896, -81.93, 97.893, 133.044]
  MoveL 1847 to (223.05, 431.25, -13.47) mm, rotated rx -180 ry 0 rz -11.91 deg; joints [23.07, -21.587, 64.91, -81.934, 97.887, 133.051]
  MoveL 1848 to (-164.9, 431.25, -13.47) mm, rotated rx -180 ry 0 rz -11.91 deg; joints [11.111, -28.491, 79.975, -90.302, 89.25, 140.615]
  Set speed (38.1 mm/s)
  MoveL 1849 to (-165.25, 432.42, -13.48) mm, rotated rx 180 ry 0 rz -11.91 deg; joints [11.092, -28.432, 79.847, -90.316, 89.237, 140.546]
  MoveL 1850 to (-164.27, 433.07, -13.48) mm, rotated rx -180 ry 0 rz -11.91 deg; joints [11.119, -28.387, 79.749, -90.294, 89.255, 140.493]
  Set speed (25.4 mm/s)
  MoveL 1851 to (-164.27, 433.07, -15.84) mm, rotated rx -180 ry 0 rz -11.91 deg; joints [11.12, -28.276, 79.723, -90.295, 89.255, 140.577]
  MoveL 1852 to (-164.27, 432.44, -16.48) mm, rotated rx -180 ry 0 rz -11.91 deg; joints [11.124, -28.281, 79.79, -90.292, 89.258, 140.64]
  Set speed (38.1 mm/s)
  MoveL 1853 to (-164.9, 431.8, -16.48) mm, rotated rx -180 ry 0 rz -11.91 deg; joints [11.108, -28.321, 79.878, -90.306, 89.248, 140.688]
  Set speed (76.2 mm/s)
  MoveL 1854 to (-194.97, 431.8, -16.47) mm, rotated rx -180 ry 0 rz -11.91 deg; joints [10.123, -28.615, 80.535, -91.086, 88.643, 141.059]
  MoveL 1855 to (-199.31, 431.8, -16.48) mm, rotated rx -180 ry 0 rz -11.91 deg; joints [9.98, -28.655, 80.624, -91.199, 88.556, 141.11]
  MoveL 1856 to (-199.79, 431.8, -16.48) mm, rotated rx 180 ry 0 rz -11.91 deg; joints [9.964, -28.66, 80.635, -91.212, 88.546, 141.116]
  MoveL 1857 to (-200.03, 431.77, -16.48) mm, rotated rx -180 ry 0 rz -11.91 deg; joints [9.957, -28.663, 80.643, -91.218, 88.542, 141.12]
  MoveL 1858 to (-200.27, 431.73, -16.47) mm, rotated rx 180 ry 0 rz -11.91 deg; joints [9.949, -28.668, 80.653, -91.224, 88.537, 141.126]
  MoveL 1859 to (-200.52, 431.67, -16.47) mm, rotated rx -180 ry 0 rz -11.91 deg; joints [9.941, -28.673, 80.665, -91.23, 88.532, 141.132]
  MoveL 1860 to (-204.13, 430.52, -16.48) mm, rotated rx -180 ry 0 rz -11.91 deg; joints [9.829, -28.766, 80.87, -91.322, 88.466, 141.246]
  MoveL 1861 to (-204.42, 430.43, -16.47) mm, rotated rx 180 ry 0 rz -11.91 deg; joints [9.82, -28.774, 80.887, -91.33, 88.46, 141.255]
  MoveL 1862 to (-204.57, 430.37, -16.48) mm, rotated rx -180 ry 0 rz -11.91 deg; joints [9.815, -28.778, 80.896, -91.333, 88.458, 141.26]
  MoveL 1863 to (-204.72, 430.31, -16.47) mm, rotated rx 180 ry 0 rz -11.91 deg; joints [9.811, -28.783, 80.907, -91.337, 88.455, 141.266]
  MoveL 1864 to (-204.86, 430.23, -16.48) mm, rotated rx -180 ry 0 rz -11.91 deg; joints [9.807, -28.788, 80.918, -91.341, 88.453, 141.272]
  MoveL 1865 to (-205.01, 430.15, -16.47) mm, rotated rx -180 ry 0 rz -11.91 deg; joints [9.802, -28.794, 80.931, -91.344, 88.45, 141.279]
  MoveL 1866 to (-205.16, 430.05, -16.48) mm, rotated rx 180 ry 0 rz -11.91 deg; joints [9.798, -28.8, 80.945, -91.348, 88.448, 141.287]
  MoveL 1867 to (-205.3, 429.94, -16.48) mm, rotated rx 180 ry 0 rz -11.91 deg; joints [9.794, -28.807, 80.96, -91.351, 88.445, 141.295]
  MoveL 1868 to (-205.53, 429.75, -16.48) mm, rotated rx 180 ry 0 rz -11.91 deg; joints [9.787, -28.82, 80.987, -91.357, 88.442, 141.31]
  MoveL 1869 to (-205.75, 429.52, -16.48) mm, rotated rx 180 ry 0 rz -11.91 deg; joints [9.781, -28.834, 81.018, -91.362, 88.438, 141.327]
  MoveL 1870 to (-205.92, 429.3, -16.48) mm, rotated rx -180 ry 0 rz -11.91 deg; joints [9.777, -28.847, 81.046, -91.366, 88.436, 141.342]
  MoveL 1871 to (-206.06, 429.09, -16.47) mm, rotated rx -180 ry 0 rz -11.91 deg; joints [9.774, -28.859, 81.073, -91.369, 88.434, 141.357]
  MoveL 1872 to (-206.14, 428.95, -16.47) mm, rotated rx -180 ry 0 rz -11.91 deg; joints [9.772, -28.867, 81.09, -91.37, 88.434, 141.367]
  MoveL 1873 to (-206.21, 428.82, -16.48) mm, rotated rx -180 ry 0 rz -11.91 deg; joints [9.77, -28.875, 81.107, -91.372, 88.433, 141.376]
  MoveL 1874 to (-206.27, 428.69, -16.48) mm, rotated rx 180 ry 0 rz -11.91 deg; joints [9.769, -28.882, 81.124, -91.373, 88.432, 141.385]
  MoveL 1875 to (-206.32, 428.55, -16.48) mm, rotated rx -180 ry 0 rz -11.91 deg; joints [9.768, -28.89, 81.141, -91.374, 88.432, 141.394]
  MoveL 1876 to (-206.37, 428.42, -16.48) mm, rotated rx -180 ry 0 rz -11.91 deg; joints [9.767, -28.898, 81.157, -91.375, 88.432, 141.403]
  MoveL 1877 to (-206.41, 428.28, -16.47) mm, rotated rx 180 ry 0 rz -11.91 deg; joints [9.767, -28.905, 81.173, -91.376, 88.432, 141.412]
  MoveL 1878 to (-206.47, 428.01, -16.47) mm, rotated rx 180 ry 0 rz -11.91 deg; joints [9.766, -28.92, 81.205, -91.377, 88.432, 141.429]
  MoveL 1879 to (-206.5, 427.77, -16.47) mm, rotated rx -180 ry 0 rz -11.91 deg; joints [9.766, -28.933, 81.234, -91.377, 88.432, 141.444]
  MoveL 1880 to (-206.52, 427.53, -16.48) mm, rotated rx -180 ry 0 rz -11.91 deg; joints [9.767, -28.946, 81.262, -91.377, 88.433, 141.46]
  MoveL 1881 to (-206.52, 427.04, -16.48) mm, rotated rx 180 ry 0 rz -11.91 deg; joints [9.77, -28.971, 81.317, -91.375, 88.435, 141.489]
  MoveL 1882 to (-206.52, 50.21, -16.48) mm, rotated rx -180 ry 0 rz -11.91 deg; joints [12.531, -44.54, 117.119, -89.197, 89.834, 161.712]
  MoveL 1883 to (-206.51, 49.73, -16.47) mm, rotated rx -180 ry 0 rz -11.91 deg; joints [12.536, -44.555, 117.158, -89.192, 89.835, 161.736]
  MoveL 1884 to (-206.48, 49.48, -16.48) mm, rotated rx -180 ry 0 rz -11.91 deg; joints [12.54, -44.563, 117.177, -89.189, 89.836, 161.747]
  MoveL 1885 to (-206.43, 49.24, -16.48) mm, rotated rx -180 ry 0 rz -11.91 deg; joints [12.544, -44.571, 117.196, -89.184, 89.837, 161.759]
  MoveL 1886 to (-206.37, 49.02, -16.47) mm, rotated rx 180 ry 0 rz -11.91 deg; joints [12.549, -44.577, 117.213, -89.18, 89.839, 161.769]
  MoveL 1887 to (-206.28, 48.8, -16.48) mm, rotated rx -180 ry 0 rz -11.91 deg; joints [12.554, -44.584, 117.23, -89.175, 89.84, 161.779]
  MoveL 1888 to (-206.18, 48.57, -16.47) mm, rotated rx 180 ry 0 rz -11.91 deg; joints [12.561, -44.591, 117.246, -89.169, 89.842, 161.789]
  MoveL 1889 to (-206.06, 48.35, -16.48) mm, rotated rx 180 ry 0 rz -11.91 deg; joints [12.568, -44.597, 117.262, -89.162, 89.844, 161.798]
  MoveL 1890 to (-205.98, 48.22, -16.48) mm, rotated rx 180 ry 0 rz -11.91 deg; joints [12.573, -44.601, 117.271, -89.157, 89.845, 161.804]
  MoveL 1891 to (-205.88, 48.09, -16.48) mm, rotated rx 180 ry 0 rz -11.91 deg; joints [12.578, -44.604, 117.28, -89.153, 89.847, 161.809]
  MoveL 1892 to (-205.78, 47.96, -16.47) mm, rotated rx -180 ry 0 rz -11.91 deg; joints [12.583, -44.608, 117.289, -89.147, 89.848, 161.814]
  MoveL 1893 to (-205.66, 47.83, -16.48) mm, rotated rx -180 ry 0 rz -11.91 deg; joints [12.589, -44.611, 117.298, -89.142, 89.85, 161.82]
  MoveL 1894 to (-205.51, 47.67, -16.48) mm, rotated rx -180 ry 0 rz -11.91 deg; joints [12.597, -44.615, 117.308, -89.134, 89.852, 161.826]
  MoveL 1895 to (-205.35, 47.54, -16.48) mm, rotated rx -180 ry 0 rz -11.91 deg; joints [12.605, -44.619, 117.316, -89.126, 89.854, 161.83]
  MoveL 1896 to (-205.19, 47.42, -16.47) mm, rotated rx 180 ry 0 rz -11.91 deg; joints [12.613, -44.622, 117.323, -89.119, 89.857, 161.835]
  MoveL 1897 to (-205.03, 47.31, -16.47) mm, rotated rx -180 ry 0 rz -11.91 deg; joints [12.621, -44.624, 117.329, -89.112, 89.859, 161.838]
  MoveL 1898 to (-204.81, 47.18, -16.47) mm, rotated rx 180 ry 0 rz -11.91 deg; joints [12.631, -44.627, 117.335, -89.102, 89.862, 161.842]
  MoveL 1899 to (-204.58, 47.08, -16.48) mm, rotated rx 180 ry 0 rz -11.91 deg; joints [12.642, -44.629, 117.34, -89.092, 89.865, 161.845]
  MoveL 1900 to (-204.36, 46.99, -16.48) mm, rotated rx 180 ry 0 rz -11.91 deg; joints [12.652, -44.63, 117.342, -89.082, 89.868, 161.846]
  MoveL 1901 to (-204.13, 46.92, -16.48) mm, rotated rx -180 ry 0 rz -11.91 deg; joints [12.662, -44.63, 117.344, -89.072, 89.871, 161.847]
  MoveL 1902 to (-203.89, 46.87, -16.48) mm, rotated rx 180 ry 0 rz -11.91 deg; joints [12.673, -44.63, 117.344, -89.062, 89.874, 161.847]
  MoveL 1903 to (-203.65, 46.84, -16.48) mm, rotated rx -180 ry 0 rz -11.91 deg; joints [12.683, -44.63, 117.342, -89.052, 89.877, 161.846]
  MoveL 1904 to (-203.41, 46.83, -16.48) mm, rotated rx -180 ry 0 rz -11.91 deg; joints [12.693, -44.629, 117.338, -89.042, 89.88, 161.844]
  MoveL 1905 to (-203.17, 46.83, -16.48) mm, rotated rx -180 ry 0 rz -11.91 deg; joints [12.703, -44.627, 117.334, -89.033, 89.883, 161.841]
  MoveL 1906 to (222.09, 46.83, -16.48) mm, rotated rx -180 ry 0 rz -11.91 deg; joints [28.86, -39.256, 103.914, -74.346, 96.845, 154.791]
  MoveL 1907 to (223.29, 46.83, -16.47) mm, rotated rx -180 ry 0 rz -11.91 deg; joints [28.901, -39.234, 103.86, -74.313, 96.87, 154.765]
  MoveL 1908 to (223.53, 46.84, -16.47) mm, rotated rx 180 ry 0 rz -11.91 deg; joints [28.909, -39.229, 103.848, -74.306, 96.875, 154.759]
  MoveL 1909 to (223.77, 46.87, -16.48) mm, rotated rx -180 ry 0 rz -11.91 deg; joints [28.916, -39.223, 103.834, -74.3, 96.88, 154.753]
  MoveL 1910 to (224.01, 46.92, -16.47) mm, rotated rx -180 ry 0 rz -11.91 deg; joints [28.923, -39.217, 103.819, -74.295, 96.885, 154.745]
  MoveL 1911 to (224.24, 46.99, -16.47) mm, rotated rx -180 ry 0 rz -11.91 deg; joints [28.93, -39.21, 103.804, -74.29, 96.89, 154.737]
  MoveL 1912 to (224.46, 47.08, -16.48) mm, rotated rx -180 ry 0 rz -11.91 deg; joints [28.936, -39.203, 103.787, -74.286, 96.896, 154.728]
  MoveL 1913 to (224.69, 47.18, -16.48) mm, rotated rx -180 ry 0 rz -11.91 deg; joints [28.941, -39.195, 103.768, -74.282, 96.901, 154.719]
  MoveL 1914 to (224.92, 47.31, -16.48) mm, rotated rx 180 ry 0 rz -11.91 deg; joints [28.946, -39.186, 103.747, -74.278, 96.906, 154.708]
  MoveL 1915 to (225.07, 47.42, -16.48) mm, rotated rx -180 ry 0 rz -11.91 deg; joints [28.95, -39.179, 103.732, -74.276, 96.91, 154.699]
  MoveL 1916 to (225.23, 47.54, -16.48) mm, rotated rx -180 ry 0 rz -11.91 deg; joints [28.953, -39.172, 103.715, -74.275, 96.914, 154.69]
  MoveL 1917 to (225.39, 47.67, -16.47) mm, rotated rx 180 ry 0 rz -11.91 deg; joints [28.956, -39.164, 103.697, -74.273, 96.918, 154.681]
  MoveL 1918 to (225.55, 47.83, -16.48) mm, rotated rx 180 ry 0 rz -11.91 deg; joints [28.958, -39.156, 103.677, -74.273, 96.922, 154.67]
  MoveL 1919 to (225.66, 47.96, -16.48) mm, rotated rx 180 ry 0 rz -11.91 deg; joints [28.959, -39.149, 103.661, -74.272, 96.925, 154.661]
  MoveL 1920 to (225.77, 48.09, -16.48) mm, rotated rx 180 ry 0 rz -11.91 deg; joints [28.96, -39.143, 103.646, -74.272, 96.928, 154.653]
  MoveL 1921 to (225.86, 48.22, -16.48) mm, rotated rx -180 ry 0 rz -11.91 deg; joints [28.961, -39.136, 103.631, -74.273, 96.93, 154.645]
  MoveL 1922 to (225.94, 48.35, -16.47) mm, rotated rx -180 ry 0 rz -11.91 deg; joints [28.962, -39.13, 103.617, -74.273, 96.933, 154.637]
  MoveL 1923 to (226.07, 48.57, -16.48) mm, rotated rx -180 ry 0 rz -11.91 deg; joints [28.961, -39.12, 103.593, -74.275, 96.936, 154.624]
  MoveL 1924 to (226.17, 48.8, -16.48) mm, rotated rx 180 ry 0 rz -11.91 deg; joints [28.961, -39.11, 103.57, -74.277, 96.939, 154.611]
  MoveL 1925 to (226.25, 49.02, -16.48) mm, rotated rx -180 ry 0 rz -11.91 deg; joints [28.959, -39.101, 103.549, -74.28, 96.942, 154.599]
  MoveL 1926 to (226.31, 49.24, -16.48) mm, rotated rx 180 ry 0 rz -11.91 deg; joints [28.957, -39.092, 103.528, -74.283, 96.945, 154.587]
  MoveL 1927 to (226.36, 49.48, -16.48) mm, rotated rx 180 ry 0 rz -11.91 deg; joints [28.954, -39.082, 103.506, -74.287, 96.947, 154.575]
  MoveL 1928 to (226.39, 49.73, -16.47) mm, rotated rx -180 ry 0 rz -11.91 deg; joints [28.951, -39.073, 103.485, -74.292, 96.949, 154.563]
  MoveL 1929 to (226.4, 50.21, -16.48) mm, rotated rx -180 ry 0 rz -11.91 deg; joints [28.942, -39.056, 103.445, -74.302, 96.951, 154.54]
  MoveL 1930 to (226.4, 428.49, -16.48) mm, rotated rx -180 ry 0 rz -11.91 deg; joints [23.201, -21.54, 65.051, -81.816, 97.955, 133.253]
  MoveL 1931 to (226.4, 428.74, -16.47) mm, rotated rx -180 ry 0 rz -11.91 deg; joints [23.198, -21.524, 65.019, -81.821, 97.955, 133.236]
  MoveL 1932 to (226.38, 428.98, -16.47) mm, rotated rx -180 ry 0 rz -11.91 deg; joints [23.195, -21.509, 64.987, -81.825, 97.955, 133.219]
  MoveL 1933 to (226.35, 429.22, -16.48) mm, rotated rx -180 ry 0 rz -11.91 deg; joints [23.191, -21.495, 64.957, -81.831, 97.954, 133.202]
  MoveL 1934 to (226.29, 429.46, -16.48) mm, rotated rx 180 ry 0 rz -11.91 deg; joints [23.186, -21.481, 64.927, -81.836, 97.953, 133.186]
  MoveL 1935 to (226.22, 429.7, -16.48) mm, rotated rx -180 ry 0 rz -11.91 deg; joints [23.181, -21.468, 64.899, -81.842, 97.952, 133.171]
  MoveL 1936 to (226.12, 429.94, -16.48) mm, rotated rx -180 ry 0 rz -11.91 deg; joints [23.175, -21.455, 64.872, -81.848, 97.949, 133.156]
  MoveL 1937 to (226.04, 430.11, -16.47) mm, rotated rx -180 ry 0 rz -11.91 deg; joints [23.171, -21.446, 64.854, -81.852, 97.948, 133.146]
  MoveL 1938 to (225.94, 430.28, -16.47) mm, rotated rx -180 ry 0 rz -11.91 deg; joints [23.166, -21.438, 64.837, -81.857, 97.945, 133.137]
  MoveL 1939 to (225.86, 430.4, -16.47) mm, rotated rx -180 ry 0 rz -11.91 deg; joints [23.162, -21.432, 64.825, -81.86, 97.944, 133.13]
  MoveL 1940 to (225.77, 430.53, -16.48) mm, rotated rx -180 ry 0 rz -11.91 deg; joints [23.158, -21.427, 64.813, -81.864, 97.941, 133.123]
  MoveL 1941 to (225.67, 430.65, -16.48) mm, rotated rx -180 ry 0 rz -11.91 deg; joints [23.154, -21.421, 64.802, -81.868, 97.939, 133.117]
  MoveL 1942 to (225.57, 430.78, -16.48) mm, rotated rx 180 ry 0 rz -11.91 deg; joints [23.149, -21.416, 64.791, -81.872, 97.937, 133.111]
  MoveL 1943 to (225.42, 430.93, -16.48) mm, rotated rx -180 ry 0 rz -11.91 deg; joints [23.143, -21.411, 64.78, -81.877, 97.933, 133.104]
  MoveL 1944 to (225.27, 431.06, -16.48) mm, rotated rx -180 ry 0 rz -11.91 deg; joints [23.137, -21.406, 64.77, -81.882, 97.93, 133.099]
  MoveL 1945 to (225.12, 431.17, -16.47) mm, rotated rx -180 ry 0 rz -11.91 deg; joints [23.132, -21.403, 64.763, -81.886, 97.926, 133.094]
  MoveL 1946 to (224.98, 431.28, -16.48) mm, rotated rx -180 ry 0 rz -11.91 deg; joints [23.126, -21.4, 64.758, -81.89, 97.923, 133.091]
  MoveL 1947 to (224.74, 431.42, -16.47) mm, rotated rx 180 ry 0 rz -11.91 deg; joints [23.118, -21.397, 64.752, -81.897, 97.917, 133.087]
  MoveL 1948 to (224.5, 431.54, -16.47) mm, rotated rx -180 ry 0 rz -11.91 deg; joints [23.109, -21.396, 64.75, -81.903, 97.911, 133.085]
  MoveL 1949 to (224.25, 431.63, -16.48) mm, rotated rx -180 ry 0 rz -11.91 deg; joints [23.101, -21.397, 64.751, -81.908, 97.905, 133.085]
  MoveL 1950 to (224.01, 431.7, -16.48) mm, rotated rx 180 ry 0 rz -11.91 deg; joints [23.093, -21.399, 64.756, -81.913, 97.899, 133.087]
  MoveL 1951 to (223.77, 431.76, -16.48) mm, rotated rx 180 ry 0 rz -11.91 deg; joints [23.086, -21.402, 64.763, -81.918, 97.893, 133.09]
  MoveL 1952 to (223.53, 431.79, -16.48) mm, rotated rx -180 ry 0 rz -11.91 deg; joints [23.079, -21.406, 64.772, -81.923, 97.887, 133.094]
  MoveL 1953 to (223.29, 431.8, -16.48) mm, rotated rx -180 ry 0 rz -11.91 deg; joints [23.071, -21.412, 64.784, -81.927, 97.881, 133.1]
  MoveL 1954 to (223.05, 431.8, -16.47) mm, rotated rx -180 ry 0 rz -11.91 deg; joints [23.065, -21.419, 64.798, -81.931, 97.875, 133.107]
  MoveL 1955 to (-164.9, 431.8, -16.48) mm, rotated rx -180 ry 0 rz -11.91 deg; joints [11.108, -28.321, 79.878, -90.306, 89.248, 140.688]
  MoveL 1956 to (-194.97, 431.99, -17.52) mm, rotated rx -180 ry 0 rz -11.91 deg; joints [10.122, -28.555, 80.501, -91.087, 88.643, 141.084]
  MoveL 1957 to (-195.47, 431.99, -17.53) mm, rotated rx -180 ry 0 rz -11.91 deg; joints [10.106, -28.56, 80.512, -91.1, 88.633, 141.09]
  MoveL 1958 to (-198.35, 431.99, -17.53) mm, rotated rx -180 ry 0 rz -11.91 deg; joints [10.011, -28.587, 80.571, -91.175, 88.575, 141.124]
  MoveL 1959 to (-199.1, 431.99, -17.53) mm, rotated rx 180 ry 0 rz -11.91 deg; joints [9.986, -28.594, 80.586, -91.195, 88.56, 141.133]
  MoveL 1960 to (-199.28, 431.98, -17.52) mm, rotated rx -180 ry 0 rz -11.91 deg; joints [9.98, -28.596, 80.592, -91.2, 88.556, 141.136]
  MoveL 1961 to (-199.47, 431.96, -17.53) mm, rotated rx 180 ry 0 rz -11.91 deg; joints [9.974, -28.599, 80.598, -91.205, 88.553, 141.14]
  MoveL 1962 to (-199.66, 431.92, -17.52) mm, rotated rx 180 ry 0 rz -11.91 deg; joints [9.968, -28.602, 80.606, -91.21, 88.549, 141.144]
  MoveL 1963 to (-199.85, 431.88, -17.53) mm, rotated rx 180 ry 0 rz -11.91 deg; joints [9.962, -28.607, 80.615, -91.214, 88.546, 141.149]
  MoveL 1964 to (-200.27, 431.74, -17.53) mm, rotated rx -180 ry 0 rz -11.91 deg; joints [9.949, -28.618, 80.639, -91.225, 88.538, 141.163]
  MoveL 1965 to (-204.13, 430.52, -17.53) mm, rotated rx 180 ry 0 rz -11.91 deg; joints [9.829, -28.717, 80.858, -91.323, 88.467, 141.284]
  MoveL 1966 to (-204.42, 430.43, -17.53) mm, rotated rx 180 ry 0 rz -11.91 deg; joints [9.82, -28.725, 80.875, -91.33, 88.461, 141.293]
  MoveL 1967 to (-204.57, 430.37, -17.52) mm, rotated rx -180 ry 0 rz -11.91 deg; joints [9.816, -28.729, 80.885, -91.334, 88.459, 141.298]
  MoveL 1968 to (-204.72, 430.31, -17.53) mm, rotated rx -180 ry 0 rz -11.91 deg; joints [9.811, -28.734, 80.895, -91.338, 88.456, 141.304]
  MoveL 1969 to (-204.86, 430.23, -17.53) mm, rotated rx -180 ry 0 rz -11.91 deg; joints [9.807, -28.739, 80.907, -91.341, 88.454, 141.31]
  MoveL 1970 to (-205.01, 430.15, -17.53) mm, rotated rx 180 ry 0 rz -11.91 deg; joints [9.802, -28.745, 80.919, -91.345, 88.451, 141.317]
  MoveL 1971 to (-205.16, 430.05, -17.52) mm, rotated rx -180 ry 0 rz -11.91 deg; joints [9.798, -28.751, 80.933, -91.349, 88.449, 141.325]
  MoveL 1972 to (-205.3, 429.94, -17.53) mm, rotated rx -180 ry 0 rz -11.91 deg; joints [9.794, -28.758, 80.948, -91.352, 88.446, 141.333]
  MoveL 1973 to (-205.53, 429.75, -17.53) mm, rotated rx -180 ry 0 rz -11.91 deg; joints [9.788, -28.77, 80.975, -91.357, 88.443, 141.348]
  MoveL 1974 to (-205.75, 429.52, -17.52) mm, rotated rx -180 ry 0 rz -11.91 deg; joints [9.782, -28.785, 81.007, -91.363, 88.44, 141.365]
  MoveL 1975 to (-205.92, 429.3, -17.52) mm, rotated rx -180 ry 0 rz -11.91 deg; joints [9.777, -28.797, 81.034, -91.367, 88.437, 141.38]
  MoveL 1976 to (-206.06, 429.09, -17.53) mm, rotated rx -180 ry 0 rz -11.91 deg; joints [9.774, -28.81, 81.062, -91.37, 88.435, 141.395]
  MoveL 1977 to (-206.14, 428.95, -17.53) mm, rotated rx -180 ry 0 rz -11.91 deg; joints [9.772, -28.818, 81.079, -91.371, 88.435, 141.404]
  MoveL 1978 to (-206.21, 428.82, -17.53) mm, rotated rx -180 ry 0 rz -11.91 deg; joints [9.771, -28.825, 81.096, -91.373, 88.434, 141.414]
  MoveL 1979 to (-206.27, 428.69, -17.53) mm, rotated rx -180 ry 0 rz -11.91 deg; joints [9.769, -28.833, 81.112, -91.374, 88.433, 141.423]
  MoveL 1980 to (-206.32, 428.55, -17.53) mm, rotated rx -180 ry 0 rz -11.91 deg; joints [9.768, -28.841, 81.129, -91.375, 88.433, 141.432]
  MoveL 1981 to (-206.37, 428.42, -17.52) mm, rotated rx -180 ry 0 rz -11.91 deg; joints [9.768, -28.848, 81.145, -91.376, 88.433, 141.441]
  MoveL 1982 to (-206.41, 428.28, -17.52) mm, rotated rx -180 ry 0 rz -11.91 deg; joints [9.767, -28.856, 81.162, -91.377, 88.433, 141.449]
  MoveL 1983 to (-206.47, 428.01, -17.52) mm, rotated rx -180 ry 0 rz -11.91 deg; joints [9.766, -28.87, 81.194, -91.377, 88.433, 141.467]
  MoveL 1984 to (-206.5, 427.77, -17.53) mm, rotated rx 180 ry 0 rz -11.91 deg; joints [9.767, -28.883, 81.222, -91.378, 88.433, 141.482]
  MoveL 1985 to (-206.52, 427.53, -17.53) mm, rotated rx -180 ry 0 rz -11.91 deg; joints [9.768, -28.896, 81.25, -91.377, 88.434, 141.497]
  MoveL 1986 to (-206.52, 427.04, -17.52) mm, rotated rx -180 ry 0 rz -11.91 deg; joints [9.77, -28.922, 81.306, -91.376, 88.437, 141.527]
  MoveL 1987 to (-206.52, 50.21, -17.52) mm, rotated rx 180 ry 0 rz -11.91 deg; joints [12.532, -44.474, 117.107, -89.196, 89.833, 161.766]
  MoveL 1988 to (-206.51, 49.73, -17.53) mm, rotated rx -180 ry 0 rz -11.91 deg; joints [12.537, -44.49, 117.147, -89.192, 89.835, 161.79]
  MoveL 1989 to (-206.48, 49.48, -17.53) mm, rotated rx 180 ry 0 rz -11.91 deg; joints [12.54, -44.498, 117.166, -89.188, 89.835, 161.801]
  MoveL 1990 to (-206.43, 49.24, -17.53) mm, rotated rx -180 ry 0 rz -11.91 deg; joints [12.545, -44.505, 117.185, -89.184, 89.837, 161.812]
  MoveL 1991 to (-206.37, 49.02, -17.53) mm, rotated rx 180 ry 0 rz -11.91 deg; joints [12.549, -44.512, 117.202, -89.18, 89.838, 161.823]
  MoveL 1992 to (-206.28, 48.8, -17.52) mm, rotated rx -180 ry 0 rz -11.91 deg; joints [12.555, -44.519, 117.219, -89.175, 89.839, 161.833]
  MoveL 1993 to (-206.18, 48.57, -17.53) mm, rotated rx -180 ry 0 rz -11.91 deg; joints [12.561, -44.525, 117.235, -89.169, 89.841, 161.843]
  MoveL 1994 to (-206.06, 48.35, -17.52) mm, rotated rx -180 ry 0 rz -11.91 deg; joints [12.568, -44.532, 117.251, -89.162, 89.843, 161.852]
  MoveL 1995 to (-205.98, 48.22, -17.53) mm, rotated rx 180 ry 0 rz -11.91 deg; joints [12.573, -44.535, 117.26, -89.157, 89.844, 161.858]
  MoveL 1996 to (-205.88, 48.09, -17.53) mm, rotated rx -180 ry 0 rz -11.91 deg; joints [12.578, -44.539, 117.269, -89.152, 89.846, 161.863]
  MoveL 1997 to (-205.78, 47.96, -17.53) mm, rotated rx -180 ry 0 rz -11.91 deg; joints [12.584, -44.543, 117.278, -89.147, 89.847, 161.868]
  MoveL 1998 to (-205.66, 47.83, -17.53) mm, rotated rx -180 ry 0 rz -11.91 deg; joints [12.59, -44.546, 117.286, -89.141, 89.849, 161.873]
  MoveL 1999 to (-205.51, 47.67, -17.53) mm, rotated rx -180 ry 0 rz -11.91 deg; joints [12.598, -44.55, 117.296, -89.134, 89.851, 161.879]
  MoveL 2000 to (-205.35, 47.54, -17.52) mm, rotated rx -180 ry 0 rz -11.91 deg; joints [12.606, -44.553, 117.305, -89.126, 89.854, 161.884]
  MoveL 2001 to (-205.19, 47.42, -17.53) mm, rotated rx -180 ry 0 rz -11.91 deg; joints [12.613, -44.556, 117.312, -89.119, 89.856, 161.889]
  MoveL 2002 to (-205.03, 47.31, -17.52) mm, rotated rx -180 ry 0 rz -11.91 deg; joints [12.621, -44.559, 117.317, -89.111, 89.858, 161.892]
  MoveL 2003 to (-204.81, 47.18, -17.53) mm, rotated rx -180 ry 0 rz -11.91 deg; joints [12.632, -44.561, 117.324, -89.101, 89.861, 161.896]
  MoveL 2004 to (-204.58, 47.08, -17.53) mm, rotated rx -180 ry 0 rz -11.91 deg; joints [12.642, -44.563, 117.328, -89.091, 89.864, 161.898]
  MoveL 2005 to (-204.36, 46.99, -17.53) mm, rotated rx -180 ry 0 rz -11.91 deg; joints [12.652, -44.564, 117.331, -89.082, 89.867, 161.9]
  MoveL 2006 to (-204.13, 46.92, -17.53) mm, rotated rx 180 ry 0 rz -11.91 deg; joints [12.662, -44.565, 117.332, -89.072, 89.87, 161.901]
  MoveL 2007 to (-203.89, 46.87, -17.52) mm, rotated rx 180 ry 0 rz -11.91 deg; joints [12.673, -44.565, 117.332, -89.062, 89.873, 161.901]
  MoveL 2008 to (-203.65, 46.84, -17.53) mm, rotated rx -180 ry 0 rz -11.91 deg; joints [12.683, -44.564, 117.33, -89.052, 89.876, 161.9]
  MoveL 2009 to (-203.41, 46.83, -17.52) mm, rotated rx 180 ry 0 rz -11.91 deg; joints [12.694, -44.563, 117.327, -89.042, 89.88, 161.897]
  MoveL 2010 to (-203.17, 46.83, -17.53) mm, rotated rx -180 ry 0 rz -11.91 deg; joints [12.704, -44.562, 117.323, -89.033, 89.883, 161.895]
  MoveL 2011 to (222.09, 46.83, -17.53) mm, rotated rx 180 ry 0 rz -11.91 deg; joints [28.861, -39.199, 103.903, -74.34, 96.832, 154.836]
  MoveL 2012 to (223.29, 46.83, -17.53) mm, rotated rx -180 ry 0 rz -11.91 deg; joints [28.901, -39.176, 103.849, -74.307, 96.857, 154.81]
  MoveL 2013 to (223.53, 46.84, -17.52) mm, rotated rx -180 ry 0 rz -11.91 deg; joints [28.909, -39.171, 103.837, -74.3, 96.863, 154.804]
  MoveL 2014 to (223.77, 46.87, -17.53) mm, rotated rx -180 ry 0 rz -11.91 deg; joints [28.917, -39.166, 103.823, -74.295, 96.868, 154.798]
  MoveL 2015 to (224.01, 46.92, -17.53) mm, rotated rx 180 ry 0 rz -11.91 deg; joints [28.924, -39.159, 103.808, -74.289, 96.873, 154.79]
  MoveL 2016 to (224.24, 46.99, -17.53) mm, rotated rx 180 ry 0 rz -11.91 deg; joints [28.93, -39.153, 103.793, -74.284, 96.878, 154.782]
  MoveL 2017 to (224.46, 47.08, -17.52) mm, rotated rx -180 ry 0 rz -11.91 deg; joints [28.936, -39.146, 103.776, -74.28, 96.883, 154.773]
  MoveL 2018 to (224.69, 47.18, -17.53) mm, rotated rx 180 ry 0 rz -11.91 deg; joints [28.942, -39.138, 103.757, -74.276, 96.888, 154.764]
  MoveL 2019 to (224.92, 47.31, -17.53) mm, rotated rx -180 ry 0 rz -11.91 deg; joints [28.947, -39.129, 103.737, -74.273, 96.894, 154.753]
  MoveL 2020 to (225.07, 47.42, -17.53) mm, rotated rx -180 ry 0 rz -11.91 deg; joints [28.95, -39.122, 103.721, -74.271, 96.898, 154.744]
  MoveL 2021 to (225.23, 47.54, -17.53) mm, rotated rx -180 ry 0 rz -11.91 deg; joints [28.953, -39.115, 103.704, -74.269, 96.901, 154.735]
  MoveL 2022 to (225.39, 47.67, -17.53) mm, rotated rx 180 ry 0 rz -11.91 deg; joints [28.956, -39.107, 103.686, -74.268, 96.905, 154.726]
  MoveL 2023 to (225.55, 47.83, -17.53) mm, rotated rx -180 ry 0 rz -11.91 deg; joints [28.958, -39.099, 103.666, -74.267, 96.91, 154.715]
  MoveL 2024 to (225.66, 47.96, -17.52) mm, rotated rx -180 ry 0 rz -11.91 deg; joints [28.96, -39.092, 103.65, -74.266, 96.913, 154.706]
  MoveL 2025 to (225.77, 48.09, -17.53) mm, rotated rx -180 ry 0 rz -11.91 deg; joints [28.961, -39.085, 103.635, -74.267, 96.915, 154.698]
  MoveL 2026 to (225.86, 48.22, -17.53) mm, rotated rx 180 ry 0 rz -11.91 deg; joints [28.962, -39.079, 103.62, -74.267, 96.918, 154.69]
  MoveL 2027 to (225.94, 48.35, -17.53) mm, rotated rx -180 ry 0 rz -11.91 deg; joints [28.962, -39.073, 103.606, -74.268, 96.92, 154.682]
  MoveL 2028 to (226.07, 48.57, -17.53) mm, rotated rx -180 ry 0 rz -11.91 deg; joints [28.962, -39.063, 103.582, -74.269, 96.924, 154.669]
  MoveL 2029 to (226.17, 48.8, -17.52) mm, rotated rx -180 ry 0 rz -11.91 deg; joints [28.961, -39.053, 103.559, -74.271, 96.927, 154.656]
  MoveL 2030 to (226.25, 49.02, -17.53) mm, rotated rx -180 ry 0 rz -11.91 deg; joints [28.96, -39.044, 103.538, -74.274, 96.93, 154.644]
  MoveL 2031 to (226.31, 49.24, -17.53) mm, rotated rx -180 ry 0 rz -11.91 deg; joints [28.958, -39.035, 103.517, -74.277, 96.932, 154.632]
  MoveL 2032 to (226.36, 49.48, -17.53) mm, rotated rx -180 ry 0 rz -11.91 deg; joints [28.955, -39.025, 103.495, -74.281, 96.934, 154.62]
  MoveL 2033 to (226.39, 49.73, -17.53) mm, rotated rx -180 ry 0 rz -11.91 deg; joints [28.951, -39.016, 103.474, -74.286, 96.936, 154.608]
  MoveL 2034 to (226.4, 50.21, -17.53) mm, rotated rx 180 ry 0 rz -11.91 deg; joints [28.943, -38.999, 103.434, -74.296, 96.939, 154.585]
  MoveL 2035 to (226.4, 428.01, -17.53) mm, rotated rx -180 ry 0 rz -11.91 deg; joints [23.208, -21.524, 65.103, -81.802, 97.95, 133.322]
  MoveL 2036 to (226.4, 428.98, -17.52) mm, rotated rx -180 ry 0 rz -11.91 deg; joints [23.196, -21.462, 64.973, -81.82, 97.951, 133.252]
  MoveL 2037 to (226.38, 429.22, -17.53) mm, rotated rx 180 ry 0 rz -11.91 deg; joints [23.192, -21.447, 64.942, -81.825, 97.95, 133.235]
  MoveL 2038 to (226.34, 429.46, -17.53) mm, rotated rx 180 ry 0 rz -11.91 deg; joints [23.188, -21.433, 64.911, -81.83, 97.95, 133.218]
  MoveL 2039 to (226.28, 429.7, -17.52) mm, rotated rx -180 ry 0 rz -11.91 deg; joints [23.183, -21.419, 64.882, -81.836, 97.949, 133.203]
  MoveL 2040 to (226.2, 429.94, -17.52) mm, rotated rx -180 ry 0 rz -11.91 deg; joints [23.178, -21.406, 64.854, -81.841, 97.947, 133.187]
  MoveL 2041 to (226.15, 430.07, -17.53) mm, rotated rx -180 ry 0 rz -11.91 deg; joints [23.175, -21.399, 64.839, -81.845, 97.946, 133.179]
  MoveL 2042 to (226.09, 430.21, -17.52) mm, rotated rx -180 ry 0 rz -11.91 deg; joints [23.172, -21.392, 64.825, -81.848, 97.944, 133.171]
  MoveL 2043 to (226.02, 430.34, -17.52) mm, rotated rx 180 ry 0 rz -11.91 deg; joints [23.168, -21.386, 64.811, -81.852, 97.943, 133.164]
  MoveL 2044 to (225.94, 430.47, -17.53) mm, rotated rx -180 ry 0 rz -11.91 deg; joints [23.164, -21.379, 64.798, -81.855, 97.941, 133.156]
  MoveL 2045 to (225.78, 430.71, -17.52) mm, rotated rx -180 ry 0 rz -11.91 deg; joints [23.156, -21.368, 64.774, -81.862, 97.937, 133.143]
  MoveL 2046 to (225.58, 430.96, -17.53) mm, rotated rx -180 ry 0 rz -11.91 deg; joints [23.148, -21.358, 64.753, -81.87, 97.933, 133.131]
  MoveL 2047 to (225.44, 431.1, -17.53) mm, rotated rx -180 ry 0 rz -11.91 deg; joints [23.142, -21.352, 64.741, -81.875, 97.929, 133.124]
  MoveL 2048 to (225.3, 431.23, -17.53) mm, rotated rx -180 ry 0 rz -11.91 deg; joints [23.136, -21.348, 64.732, -81.88, 97.926, 133.119]
  MoveL 2049 to (225.16, 431.34, -17.53) mm, rotated rx -180 ry 0 rz -11.91 deg; joints [23.131, -21.344, 64.725, -81.884, 97.923, 133.115]
  MoveL 2050 to (225.02, 431.44, -17.53) mm, rotated rx -180 ry 0 rz -11.91 deg; joints [23.126, -21.342, 64.719, -81.888, 97.919, 133.111]
  MoveL 2051 to (224.78, 431.59, -17.53) mm, rotated rx 180 ry 0 rz -11.91 deg; joints [23.117, -21.339, 64.713, -81.894, 97.914, 133.107]
